LIN {X 116.831,Y -35.719,Z -65.842,A -90.000,B 90.000,C 0.000} C_DIS
LIN {X 116.119,Y -35.719,Z -68.117,A -90.000,B 90.000,C 0.000} C_DIS
LIN {X 115.340,Y -35.719,Z -70.370,A -90.000,B 90.000,C 0.000} C_DIS
LIN {X 114.495,Y -35.719,Z -72.600,A -90.000,B 90.000,C 0.000} C_DIS
LIN {X 113.585,Y -35.719,Z -74.804,A -90.000,B 90.000,C 0.000} C_DIS
LIN {X 112.611,Y -35.719,Z -76.980,A -90.000,B 90.000,C 0.000} C_DIS
LIN {X 111.574,Y -35.719,Z -79.127,A -90.000,B 90.000,C 0.000} C_DIS
LIN {X 110.474,Y -35.719,Z -81.243,A -90.000,B 90.000,C 0.000} C_DIS
LIN {X 109.313,Y -35.719,Z -83.325,A -90.000,B 90.000,C 0.000} C_DIS
LIN {X 108.091,Y -35.719,Z -85.373,A -90.000,B 90.000,C 0.000} C_DIS
LIN {X 106.810,Y -35.719,Z -87.384,A -90.000,B 90.000,C 0.000} C_DIS
LIN {X 105.470,Y -35.719,Z -89.356,A -90.000,B 90.000,C 0.000} C_DIS
LIN {X 105.415,Y -35.719,Z -90.221,A -90.000,B 90.000,C 0.000} C_DIS
LIN {X 105.339,Y -35.719,Z -91.084,A -90.000,B 90.000,C 0.000} C_DIS
LIN {X 105.322,Y -35.719,Z -92.275,A -90.000,B 90.000,C 0.000} C_DIS
LIN {X 105.256,Y -35.719,Z -93.465,A -90.000,B 90.000,C 0.000} C_DIS
LIN {X 105.138,Y -35.719,Z -94.651,A -90.000,B 90.000,C 0.000} C_DIS
LIN {X 104.971,Y -35.719,Z -95.830,A -90.000,B 90.000,C 0.000} C_DIS
LIN {X 104.754,Y -35.719,Z -97.002,A -90.000,B 90.000,C 0.000} C_DIS
LIN {X 104.487,Y -35.719,Z -98.163,A -90.000,B 90.000,C 0.000} C_DIS
LIN {X 104.172,Y -35.719,Z -99.312,A -90.000,B 90.000,C 0.000} C_DIS
LIN {X 103.843,Y -35.719,Z -100.216,A -90.000,B 90.000,C 0.000} C_DIS
LIN {X 103.553,Y -35.719,Z -101.134,A -90.000,B 90.000,C 0.000} C_DIS
LIN {X 103.303,Y -35.719,Z -102.064,A -90.000,B 90.000,C 0.000} C_DIS
LIN {X 103.095,Y -35.719,Z -103.004,A -90.000,B 90.000,C 0.000} C_DIS
LIN {X 102.892,Y -35.719,Z -103.459,A -90.000,B 90.000,C 0.000} C_DIS
LIN {X 102.749,Y -35.719,Z -103.936,A -90.000,B 90.000,C 0.000} C_DIS
LIN {X 102.667,Y -35.719,Z -104.427,A -90.000,B 90.000,C 0.000} C_DIS
LIN {X 102.649,Y -35.719,Z -104.925,A -90.000,B 90.000,C 0.000} C_DIS
LIN {X 102.693,Y -35.719,Z -105.421,A -90.000,B 90.000,C 0.000} C_DIS
LIN {X 102.800,Y -35.719,Z -105.907,A -90.000,B 90.000,C 0.000} C_DIS
LIN {X 102.981,Y -35.719,Z -108.478,A -90.000,B 90.000,C 0.000} C_DIS
LIN {X 103.102,Y -35.719,Z -111.053,A -90.000,B 90.000,C 0.000} C_DIS
LIN {X 103.163,Y -35.719,Z -113.630,A -90.000,B 90.000,C 0.000} C_DIS
LIN {X 103.164,Y -35.719,Z -116.208,A -90.000,B 90.000,C 0.000} C_DIS
LIN {X 103.250,Y -35.719,Z -118.970,A -90.000,B 90.000,C 0.000} C_DIS
LIN {X 103.278,Y -35.719,Z -121.732,A -90.000,B 90.000,C 0.000} C_DIS
LIN {X 103.247,Y -35.719,Z -124.495,A -90.000,B 90.000,C 0.000} C_DIS
LIN {X 103.157,Y -35.719,Z -127.257,A -90.000,B 90.000,C 0.000} C_DIS
LIN {X 103.009,Y -35.719,Z -130.016,A -90.000,B 90.000,C 0.000} C_DIS
LIN {X 102.803,Y -35.719,Z -132.771,A -90.000,B 90.000,C 0.000} C_DIS
LIN {X 102.538,Y -35.719,Z -135.521,A -90.000,B 90.000,C 0.000} C_DIS
LIN {X 102.366,Y -35.719,Z -138.398,A -90.000,B 90.000,C 0.000} C_DIS
LIN {X 102.141,Y -35.719,Z -141.271,A -90.000,B 90.000,C 0.000} C_DIS
LIN {X 101.862,Y -35.719,Z -144.140,A -90.000,B 90.000,C 0.000} C_DIS
LIN {X 101.529,Y -35.719,Z -147.003,A -90.000,B 90.000,C 0.000} C_DIS
LIN {X 101.143,Y -35.719,Z -149.859,A -90.000,B 90.000,C 0.000} C_DIS
LIN {X 100.704,Y -35.719,Z -152.708,A -90.000,B 90.000,C 0.000} C_DIS
LIN {X 100.212,Y -35.719,Z -155.548,A -90.000,B 90.000,C 0.000} C_DIS
LIN {X 99.667,Y -35.719,Z -158.378,A -90.000,B 90.000,C 0.000} C_DIS
LIN {X 98.834,Y -35.719,Z -161.929,A -90.000,B 90.000,C 0.000} C_DIS
LIN {X 97.948,Y -35.719,Z -165.466,A -90.000,B 90.000,C 0.000} C_DIS
LIN {X 97.008,Y -35.719,Z -168.990,A -90.000,B 90.000,C 0.000} C_DIS
LIN {X 96.014,Y -35.719,Z -172.499,A -90.000,B 90.000,C 0.000} C_DIS
LIN {X 94.967,Y -35.719,Z -175.992,A -90.000,B 90.000,C 0.000} C_DIS
LIN {X 93.867,Y -35.719,Z -179.469,A -90.000,B 90.000,C 0.000} C_DIS
LIN {X 89.622,Y -35.719,Z -192.770,A -90.000,B 90.000,C 0.000} C_DIS
LIN {X 88.034,Y -35.719,Z -197.593,A -90.000,B 90.000,C 0.000} C_DIS
LIN {X 86.382,Y -35.719,Z -202.396,A -90.000,B 90.000,C 0.000} C_DIS
LIN {X 84.667,Y -35.719,Z -207.176,A -90.000,B 90.000,C 0.000} C_DIS
LIN {X 82.889,Y -35.719,Z -211.933,A -90.000,B 90.000,C 0.000} C_DIS
LIN {X 81.049,Y -35.719,Z -216.666,A -90.000,B 90.000,C 0.000} C_DIS
LIN {X 79.146,Y -35.719,Z -221.374,A -90.000,B 90.000,C 0.000} C_DIS
LIN {X 76.777,Y -35.719,Z -226.893,A -90.000,B 90.000,C 0.000} C_DIS
LIN {X 74.453,Y -35.719,Z -232.431,A -90.000,B 90.000,C 0.000} C_DIS
LIN {X 72.173,Y -35.719,Z -237.987,A -90.000,B 90.000,C 0.000} C_DIS
LIN {X 69.938,Y -35.719,Z -243.561,A -90.000,B 90.000,C 0.000} C_DIS
LIN {X 145.015,Y -35.719,Z -243.561,A -90.000,B 90.000,C 0.000} C_DIS
LIN {X 145.015,Y -35.719,Z 0.000,A -90.000,B 90.000,C 0.000} C_DIS
LIN {X -145.015,Y -35.719,Z 0.000,A -90.000,B 90.000,C 0.000} C_DIS
LIN {X -145.015,Y -35.719,Z -243.561,A -90.000,B 90.000,C 0.000} C_DIS
LIN {X -110.096,Y -35.719,Z -243.561,A -90.000,B 90.000,C 0.000} C_DIS
LIN {X -107.153,Y -35.719,Z -241.272,A -90.000,B 90.000,C 0.000} C_DIS
LIN {X -104.176,Y -35.719,Z -239.027,A -90.000,B 90.000,C 0.000} C_DIS
LIN {X -101.166,Y -35.719,Z -236.828,A -90.000,B 90.000,C 0.000} C_DIS
LIN {X -98.123,Y -35.719,Z -234.673,A -90.000,B 90.000,C 0.000} C_DIS
LIN {X -95.049,Y -35.719,Z -232.564,A -90.000,B 90.000,C 0.000} C_DIS
LIN {X -91.943,Y -35.719,Z -230.501,A -90.000,B 90.000,C 0.000} C_DIS
LIN {X -88.807,Y -35.719,Z -228.485,A -90.000,B 90.000,C 0.000} C_DIS
LIN {X -86.159,Y -35.719,Z -226.746,A -90.000,B 90.000,C 0.000} C_DIS
LIN {X -81.987,Y -35.719,Z -224.226,A -90.000,B 90.000,C 0.000} C_DIS
LIN {X -77.783,Y -35.719,Z -221.761,A -90.000,B 90.000,C 0.000} C_DIS
LIN {X -73.548,Y -35.719,Z -219.350,A -90.000,B 90.000,C 0.000} C_DIS
LIN {X -69.281,Y -35.719,Z -216.994,A -90.000,B 90.000,C 0.000} C_DIS
LIN {X -64.985,Y -35.719,Z -214.693,A -90.000,B 90.000,C 0.000} C_DIS
LIN {X -60.659,Y -35.719,Z -212.448,A -90.000,B 90.000,C 0.000} C_DIS
LIN {X -56.305,Y -35.719,Z -210.259,A -90.000,B 90.000,C 0.000} C_DIS
LIN {X -51.922,Y -35.719,Z -208.127,A -90.000,B 90.000,C 0.000} C_DIS
LIN {X -46.937,Y -35.719,Z -205.632,A -90.000,B 90.000,C 0.000} C_DIS
LIN {X -44.461,Y -35.719,Z -204.434,A -90.000,B 90.000,C 0.000} C_DIS
LIN {X -42.009,Y -35.719,Z -203.189,A -90.000,B 90.000,C 0.000} C_DIS
LIN {X -39.581,Y -35.719,Z -201.895,A -90.000,B 90.000,C 0.000} C_DIS
LIN {X -37.180,Y -35.719,Z -200.555,A -90.000,B 90.000,C 0.000} C_DIS
LIN {X -34.804,Y -35.719,Z -199.168,A -90.000,B 90.000,C 0.000} C_DIS
LIN {X -32.457,Y -35.719,Z -197.735,A -90.000,B 90.000,C 0.000} C_DIS
LIN {X -30.138,Y -35.719,Z -196.256,A -90.000,B 90.000,C 0.000} C_DIS
LIN {X -27.848,Y -35.719,Z -194.732,A -90.000,B 90.000,C 0.000} C_DIS
LIN {X -24.879,Y -35.719,Z -192.551,A -90.000,B 90.000,C 0.000} C_DIS
LIN {X -21.945,Y -35.719,Z -190.324,A -90.000,B 90.000,C 0.000} C_DIS
LIN {X -19.046,Y -35.719,Z -188.051,A -90.000,B 90.000,C 0.000} C_DIS
LIN {X -16.183,Y -35.719,Z -185.732,A -90.000,B 90.000,C 0.000} C_DIS
LIN {X -13.358,Y -35.719,Z -183.368,A -90.000,B 90.000,C 0.000} C_DIS
LIN {X -10.570,Y -35.719,Z -180.960,A -90.000,B 90.000,C 0.000} C_DIS
LIN {X -7.820,Y -35.719,Z -178.509,A -90.000,B 90.000,C 0.000} C_DIS
LIN {X -5.995,Y -35.719,Z -176.907,A -90.000,B 90.000,C 0.000} C_DIS
LIN {X -4.209,Y -35.719,Z -175.263,A -90.000,B 90.000,C 0.000} C_DIS
LIN {X -2.461,Y -35.719,Z -173.577,A -90.000,B 90.000,C 0.000} C_DIS
LIN {X -0.754,Y -35.719,Z -171.851,A -90.000,B 90.000,C 0.000} C_DIS
LIN {X 0.913,Y -35.719,Z -170.085,A -90.000,B 90.000,C 0.000} C_DIS
LIN {X 1.496,Y -35.719,Z -169.467,A -90.000,B 90.000,C 0.000} C_DIS
LIN {X 2.036,Y -35.719,Z -168.811,A -90.000,B 90.000,C 0.000} C_DIS
LIN {X 2.530,Y -35.719,Z -168.120,A -90.000,B 90.000,C 0.000} C_DIS
LIN {X 2.976,Y -35.719,Z -167.397,A -90.000,B 90.000,C 0.000} C_DIS
LIN {X 3.229,Y -35.719,Z -167.142,A -90.000,B 90.000,C 0.000} C_DIS
LIN {X 3.431,Y -35.719,Z -166.845,A -90.000,B 90.000,C 0.000} C_DIS
LIN {X 3.574,Y -35.719,Z -166.515,A -90.000,B 90.000,C 0.000} C_DIS
LIN {X 3.653,Y -35.719,Z -166.164,A -90.000,B 90.000,C 0.000} C_DIS
LIN {X 3.666,Y -35.719,Z -165.805,A -90.000,B 90.000,C 0.000} C_DIS
LIN {X 3.612,Y -35.719,Z -165.450,A -90.000,B 90.000,C 0.000} C_DIS
LIN {X 3.493,Y -35.719,Z -165.111,A -90.000,B 90.000,C 0.000} C_DIS
LIN {X 3.313,Y -35.719,Z -164.800,A -90.000,B 90.000,C 0.000} C_DIS
LIN {X 3.078,Y -35.719,Z -164.528,A -90.000,B 90.000,C 0.000} C_DIS
LIN {X 2.322,Y -35.719,Z -164.113,A -90.000,B 90.000,C 0.000} C_DIS
LIN {X 1.554,Y -35.719,Z -163.721,A -90.000,B 90.000,C 0.000} C_DIS
LIN {X -1.251,Y -35.719,Z -162.907,A -90.000,B 90.000,C 0.000} C_DIS
LIN {X -2.477,Y -35.719,Z -162.410,A -90.000,B 90.000,C 0.000} C_DIS
LIN {X -3.719,Y -35.719,Z -161.957,A -90.000,B 90.000,C 0.000} C_DIS
LIN {X -4.976,Y -35.719,Z -161.547,A -90.000,B 90.000,C 0.000} C_DIS
LIN {X -6.247,Y -35.719,Z -161.182,A -90.000,B 90.000,C 0.000} C_DIS
LIN {X -8.359,Y -35.719,Z -160.357,A -90.000,B 90.000,C 0.000} C_DIS
LIN {X -10.450,Y -35.719,Z -159.479,A -90.000,B 90.000,C 0.000} C_DIS
LIN {X -12.518,Y -35.719,Z -158.548,A -90.000,B 90.000,C 0.000} C_DIS
LIN {X -14.562,Y -35.719,Z -157.566,A -90.000,B 90.000,C 0.000} C_DIS
LIN {X -16.580,Y -35.719,Z -156.532,A -90.000,B 90.000,C 0.000} C_DIS
LIN {X -18.572,Y -35.719,Z -155.448,A -90.000,B 90.000,C 0.000} C_DIS
LIN {X -20.770,Y -35.719,Z -154.028,A -90.000,B 90.000,C 0.000} C_DIS
LIN {X -22.940,Y -35.719,Z -152.565,A -90.000,B 90.000,C 0.000} C_DIS
LIN {X -25.081,Y -35.719,Z -151.060,A -90.000,B 90.000,C 0.000} C_DIS
LIN {X -27.192,Y -35.719,Z -149.513,A -90.000,B 90.000,C 0.000} C_DIS
LIN {X -28.258,Y -35.719,Z -148.710,A -90.000,B 90.000,C 0.000} C_DIS
LIN {X -29.291,Y -35.719,Z -147.865,A -90.000,B 90.000,C 0.000} C_DIS
LIN {X -30.291,Y -35.719,Z -146.981,A -90.000,B 90.000,C 0.000} C_DIS
LIN {X -31.255,Y -35.719,Z -146.058,A -90.000,B 90.000,C 0.000} C_DIS
LIN {X -32.182,Y -35.719,Z -145.098,A -90.000,B 90.000,C 0.000} C_DIS
LIN {X -33.529,Y -35.719,Z -143.805,A -90.000,B 90.000,C 0.000} C_DIS
LIN {X -34.823,Y -35.719,Z -142.460,A -90.000,B 90.000,C 0.000} C_DIS
LIN {X -36.063,Y -35.719,Z -141.064,A -90.000,B 90.000,C 0.000} C_DIS
LIN {X -37.246,Y -35.719,Z -139.620,A -90.000,B 90.000,C 0.000} C_DIS
LIN {X -38.372,Y -35.719,Z -138.130,A -90.000,B 90.000,C 0.000} C_DIS
LIN {X -39.437,Y -35.719,Z -136.597,A -90.000,B 90.000,C 0.000} C_DIS
LIN {X -40.440,Y -35.719,Z -135.022,A -90.000,B 90.000,C 0.000} C_DIS
LIN {X -41.380,Y -35.719,Z -133.409,A -90.000,B 90.000,C 0.000} C_DIS
LIN {X -42.255,Y -35.719,Z -131.760,A -90.000,B 90.000,C 0.000} C_DIS
LIN {X -43.063,Y -35.719,Z -130.077,A -90.000,B 90.000,C 0.000} C_DIS
LIN {X -43.805,Y -35.719,Z -128.364,A -90.000,B 90.000,C 0.000} C_DIS
LIN {X -44.477,Y -35.719,Z -126.622,A -90.000,B 90.000,C 0.000} C_DIS
LIN {X -45.080,Y -35.719,Z -124.855,A -90.000,B 90.000,C 0.000} C_DIS
LIN {X -45.612,Y -35.719,Z -123.065,A -90.000,B 90.000,C 0.000} C_DIS
LIN {X -46.072,Y -35.719,Z -121.256,A -90.000,B 90.000,C 0.000} C_DIS
LIN {X -46.455,Y -35.719,Z -119.310,A -90.000,B 90.000,C 0.000} C_DIS
LIN {X -46.782,Y -35.719,Z -117.354,A -90.000,B 90.000,C 0.000} C_DIS
LIN {X -47.053,Y -35.719,Z -115.390,A -90.000,B 90.000,C 0.000} C_DIS
LIN {X -47.268,Y -35.719,Z -113.418,A -90.000,B 90.000,C 0.000} C_DIS
LIN {X -47.426,Y -35.719,Z -111.441,A -90.000,B 90.000,C 0.000} C_DIS
LIN {X -47.529,Y -35.719,Z -109.461,A -90.000,B 90.000,C 0.000} C_DIS
LIN {X -47.947,Y -35.719,Z -108.832,A -90.000,B 90.000,C 0.000} C_DIS
LIN {X -48.399,Y -35.719,Z -108.227,A -90.000,B 90.000,C 0.000} C_DIS
LIN {X -48.883,Y -35.719,Z -107.647,A -90.000,B 90.000,C 0.000} C_DIS
LIN {X -50.094,Y -35.719,Z -106.124,A -90.000,B 90.000,C 0.000} C_DIS
LIN {X -51.246,Y -35.719,Z -104.556,A -90.000,B 90.000,C 0.000} C_DIS
LIN {X -52.339,Y -35.719,Z -102.947,A -90.000,B 90.000,C 0.000} C_DIS
LIN {X -53.372,Y -35.719,Z -101.298,A -90.000,B 90.000,C 0.000} C_DIS
LIN {X -54.341,Y -35.719,Z -99.611,A -90.000,B 90.000,C 0.000} C_DIS
LIN {X -55.247,Y -35.719,Z -97.889,A -90.000,B 90.000,C 0.000} C_DIS
LIN {X -56.088,Y -35.719,Z -96.135,A -90.000,B 90.000,C 0.000} C_DIS
LIN {X -56.863,Y -35.719,Z -94.350,A -90.000,B 90.000,C 0.000} C_DIS
LIN {X -57.570,Y -35.719,Z -92.538,A -90.000,B 90.000,C 0.000} C_DIS
LIN {X -58.209,Y -35.719,Z -90.700,A -90.000,B 90.000,C 0.000} C_DIS
LIN {X -58.779,Y -35.719,Z -88.840,A -90.000,B 90.000,C 0.000} C_DIS
LIN {X -59.279,Y -35.719,Z -86.960,A -90.000,B 90.000,C 0.000} C_DIS
LIN {X -59.708,Y -35.719,Z -85.062,A -90.000,B 90.000,C 0.000} C_DIS
LIN {X -60.066,Y -35.719,Z -83.149,A -90.000,B 90.000,C 0.000} C_DIS
LIN {X -60.352,Y -35.719,Z -81.225,A -90.000,B 90.000,C 0.000} C_DIS
LIN {X -60.530,Y -35.719,Z -79.874,A -90.000,B 90.000,C 0.000} C_DIS
LIN {X -60.643,Y -35.719,Z -78.516,A -90.000,B 90.000,C 0.000} C_DIS
LIN {X -60.688,Y -35.719,Z -77.155,A -90.000,B 90.000,C 0.000} C_DIS
LIN {X -60.667,Y -35.719,Z -75.792,A -90.000,B 90.000,C 0.000} C_DIS
LIN {X -60.578,Y -35.719,Z -74.433,A -90.000,B 90.000,C 0.000} C_DIS
LIN {X -60.424,Y -35.719,Z -73.079,A -90.000,B 90.000,C 0.000} C_DIS
LIN {X -60.203,Y -35.719,Z -71.734,A -90.000,B 90.000,C 0.000} C_DIS
LIN {X -59.916,Y -35.719,Z -70.402,A -90.000,B 90.000,C 0.000} C_DIS
LIN {X -59.565,Y -35.719,Z -69.086,A -90.000,B 90.000,C 0.000} C_DIS
LIN {X -59.313,Y -35.719,Z -68.078,A -90.000,B 90.000,C 0.000} C_DIS
LIN {X -58.993,Y -35.719,Z -67.089,A -90.000,B 90.000,C 0.000} C_DIS
LIN {X -58.606,Y -35.719,Z -66.124,A -90.000,B 90.000,C 0.000} C_DIS
LIN {X -58.155,Y -35.719,Z -65.188,A -90.000,B 90.000,C 0.000} C_DIS
LIN {X -57.640,Y -35.719,Z -64.284,A -90.000,B 90.000,C 0.000} C_DIS
LIN {X -57.066,Y -35.719,Z -63.418,A -90.000,B 90.000,C 0.000} C_DIS
LIN {X -56.434,Y -35.719,Z -62.593,A -90.000,B 90.000,C 0.000} C_DIS
LIN {X -55.747,Y -35.719,Z -61.813,A -90.000,B 90.000,C 0.000} C_DIS
LIN {X -55.009,Y -35.719,Z -61.081,A -90.000,B 90.000,C 0.000} C_DIS
LIN {X -54.222,Y -35.719,Z -60.402,A -90.000,B 90.000,C 0.000} C_DIS
LIN {X -53.391,Y -35.719,Z -59.777,A -90.000,B 90.000,C 0.000} C_DIS
LIN {X -52.520,Y -35.719,Z -59.210,A -90.000,B 90.000,C 0.000} C_DIS
LIN {X -51.321,Y -35.719,Z -58.559,A -90.000,B 90.000,C 0.000} C_DIS
LIN {X -50.096,Y -35.719,Z -57.960,A -90.000,B 90.000,C 0.000} C_DIS
LIN {X -48.846,Y -35.719,Z -57.414,A -90.000,B 90.000,C 0.000} C_DIS
LIN {X -47.573,Y -35.719,Z -56.922,A -90.000,B 90.000,C 0.000} C_DIS
LIN {X -46.281,Y -35.719,Z -56.485,A -90.000,B 90.000,C 0.000} C_DIS
LIN {X -44.691,Y -35.719,Z -56.129,A -90.000,B 90.000,C 0.000} C_DIS
LIN {X -43.088,Y -35.719,Z -55.836,A -90.000,B 90.000,C 0.000} C_DIS
LIN {X -41.475,Y -35.719,Z -55.608,A -90.000,B 90.000,C 0.000} C_DIS
LIN {X -39.854,Y -35.719,Z -55.444,A -90.000,B 90.000,C 0.000} C_DIS
LIN {X -38.227,Y -35.719,Z -55.345,A -90.000,B 90.000,C 0.000} C_DIS
LIN {X -36.598,Y -35.719,Z -55.310,A -90.000,B 90.000,C 0.000} C_DIS
LIN {X -34.969,Y -35.719,Z -55.340,A -90.000,B 90.000,C 0.000} C_DIS
LIN {X -33.343,Y -35.719,Z -55.435,A -90.000,B 90.000,C 0.000} C_DIS
LIN {X -31.721,Y -35.719,Z -55.595,A -90.000,B 90.000,C 0.000} C_DIS
LIN {X -30.107,Y -35.719,Z -55.819,A -90.000,B 90.000,C 0.000} C_DIS
LIN {X -28.504,Y -35.719,Z -56.107,A -90.000,B 90.000,C 0.000} C_DIS
LIN {X -26.913,Y -35.719,Z -56.459,A -90.000,B 90.000,C 0.000} C_DIS
LIN {X -25.337,Y -35.719,Z -56.874,A -90.000,B 90.000,C 0.000} C_DIS
LIN {X -25.206,Y -35.719,Z -56.732,A -90.000,B 90.000,C 0.000} C_DIS
LIN {X -24.358,Y -35.719,Z -56.061,A -90.000,B 90.000,C 0.000} C_DIS
LIN {X -23.471,Y -35.719,Z -55.444,A -90.000,B 90.000,C 0.000} C_DIS
LIN {X -22.548,Y -35.719,Z -54.882,A -90.000,B 90.000,C 0.000} C_DIS
LIN {X -21.592,Y -35.719,Z -54.378,A -90.000,B 90.000,C 0.000} C_DIS
LIN {X -20.607,Y -35.719,Z -53.933,A -90.000,B 90.000,C 0.000} C_DIS
LIN {X -19.596,Y -35.719,Z -53.549,A -90.000,B 90.000,C 0.000} C_DIS
LIN {X -18.564,Y -35.719,Z -53.229,A -90.000,B 90.000,C 0.000} C_DIS
LIN {X -17.514,Y -35.719,Z -52.972,A -90.000,B 90.000,C 0.000} C_DIS
LIN {X -16.196,Y -35.719,Z -52.825,A -90.000,B 90.000,C 0.000} C_DIS
LIN {X -14.873,Y -35.719,Z -52.731,A -90.000,B 90.000,C 0.000} C_DIS
LIN {X -13.548,Y -35.719,Z -52.688,A -90.000,B 90.000,C 0.000} C_DIS
LIN {X -12.222,Y -35.719,Z -52.697,A -90.000,B 90.000,C 0.000} C_DIS
LIN {X -10.897,Y -35.719,Z -52.757,A -90.000,B 90.000,C 0.000} C_DIS
LIN {X -9.576,Y -35.719,Z -52.870,A -90.000,B 90.000,C 0.000} C_DIS
LIN {X -8.260,Y -35.719,Z -53.034,A -90.000,B 90.000,C 0.000} C_DIS
LIN {X -4.666,Y -35.719,Z -53.602,A -90.000,B 90.000,C 0.000} C_DIS
LIN {X -1.066,Y -35.719,Z -54.121,A -90.000,B 90.000,C 0.000} C_DIS
LIN {X 2.542,Y -35.719,Z -54.591,A -90.000,B 90.000,C 0.000} C_DIS
LIN {X 2.542,Y -48.219,Z -54.591,A -90.000,B 90.000,C 0.000} C_DIS
LIN {X 2.542,Y -60.719,Z -54.591,A -90.000,B 90.000,C 0.000} C_DIS
LIN {X 90.609,Y -60.719,Z -242.561,A -90.000,B 90.000,C 0.000} C_DIS
LIN {X 90.609,Y -53.575,Z -242.561,A -90.000,B 90.000,C 0.000} C_DIS
LIN {X 90.609,Y -41.075,Z -242.561,A -90.000,B 90.000,C 0.000} C_DIS
LIN {X 90.609,Y -28.575,Z -242.561,A -90.000,B 90.000,C 0.000} C_DIS
LIN {X 144.015,Y -28.575,Z -242.561,A -90.000,B 90.000,C 0.000} C_DIS
LIN {X 144.015,Y -28.575,Z -235.012,A -90.000,B 90.000,C 0.000} C_DIS
LIN {X 92.953,Y -28.575,Z -235.012,A -90.000,B 90.000,C 0.000} C_DIS
LIN {X 93.660,Y -28.575,Z -232.505,A -90.000,B 90.000,C 0.000} C_DIS
LIN {X 94.335,Y -28.575,Z -229.989,A -90.000,B 90.000,C 0.000} C_DIS
LIN {X 94.978,Y -28.575,Z -227.464,A -90.000,B 90.000,C 0.000} C_DIS
LIN {X 144.015,Y -28.575,Z -227.464,A -90.000,B 90.000,C 0.000} C_DIS
LIN {X 144.015,Y -28.575,Z -219.915,A -90.000,B 90.000,C 0.000} C_DIS
LIN {X 96.864,Y -28.575,Z -219.915,A -90.000,B 90.000,C 0.000} C_DIS
LIN {X 97.478,Y -28.575,Z -217.548,A -90.000,B 90.000,C 0.000} C_DIS
LIN {X 98.098,Y -28.575,Z -215.183,A -90.000,B 90.000,C 0.000} C_DIS
LIN {X 98.477,Y -28.575,Z -213.776,A -90.000,B 90.000,C 0.000} C_DIS
LIN {X 98.848,Y -28.575,Z -212.366,A -90.000,B 90.000,C 0.000} C_DIS
LIN {X 144.015,Y -28.575,Z -212.366,A -90.000,B 90.000,C 0.000} C_DIS
LIN {X 144.015,Y -28.575,Z -204.817,A -90.000,B 90.000,C 0.000} C_DIS
LIN {X 100.664,Y -28.575,Z -204.817,A -90.000,B 90.000,C 0.000} C_DIS
LIN {X 101.185,Y -28.575,Z -202.411,A -90.000,B 90.000,C 0.000} C_DIS
LIN {X 101.679,Y -28.575,Z -200.000,A -90.000,B 90.000,C 0.000} C_DIS
LIN {X 102.147,Y -28.575,Z -197.583,A -90.000,B 90.000,C 0.000} C_DIS
LIN {X 102.190,Y -28.575,Z -197.269,A -90.000,B 90.000,C 0.000} C_DIS
LIN {X 144.015,Y -28.575,Z -197.269,A -90.000,B 90.000,C 0.000} C_DIS
LIN {X 144.015,Y -28.575,Z -189.720,A -90.000,B 90.000,C 0.000} C_DIS
LIN {X 102.994,Y -28.575,Z -189.720,A -90.000,B 90.000,C 0.000} C_DIS
LIN {X 103.117,Y -28.575,Z -188.042,A -90.000,B 90.000,C 0.000} C_DIS
LIN {X 103.220,Y -28.575,Z -186.362,A -90.000,B 90.000,C 0.000} C_DIS
LIN {X 103.302,Y -28.575,Z -184.681,A -90.000,B 90.000,C 0.000} C_DIS
LIN {X 103.398,Y -28.575,Z -183.426,A -90.000,B 90.000,C 0.000} C_DIS
LIN {X 103.504,Y -28.575,Z -182.171,A -90.000,B 90.000,C 0.000} C_DIS
LIN {X 144.015,Y -28.575,Z -182.171,A -90.000,B 90.000,C 0.000} C_DIS
LIN {X 144.015,Y -28.575,Z -174.622,A -90.000,B 90.000,C 0.000} C_DIS
LIN {X 104.367,Y -28.575,Z -174.622,A -90.000,B 90.000,C 0.000} C_DIS
LIN {X 104.655,Y -28.575,Z -172.656,A -90.000,B 90.000,C 0.000} C_DIS
LIN {X 104.969,Y -28.575,Z -170.694,A -90.000,B 90.000,C 0.000} C_DIS
LIN {X 105.308,Y -28.575,Z -168.736,A -90.000,B 90.000,C 0.000} C_DIS
LIN {X 105.494,Y -28.575,Z -167.073,A -90.000,B 90.000,C 0.000} C_DIS
LIN {X 144.015,Y -28.575,Z -167.073,A -90.000,B 90.000,C 0.000} C_DIS
LIN {X 144.015,Y -28.575,Z -159.525,A -90.000,B 90.000,C 0.000} C_DIS
LIN {X 106.509,Y -28.575,Z -159.525,A -90.000,B 90.000,C 0.000} C_DIS
LIN {X 106.823,Y -28.575,Z -157.546,A -90.000,B 90.000,C 0.000} C_DIS
LIN {X 107.130,Y -28.575,Z -154.760,A -90.000,B 90.000,C 0.000} C_DIS
LIN {X 107.450,Y -28.575,Z -151.976,A -90.000,B 90.000,C 0.000} C_DIS
LIN {X 144.015,Y -28.575,Z -151.976,A -90.000,B 90.000,C 0.000} C_DIS
LIN {X 144.015,Y -28.575,Z -144.427,A -90.000,B 90.000,C 0.000} C_DIS
LIN {X 108.180,Y -28.575,Z -144.427,A -90.000,B 90.000,C 0.000} C_DIS
LIN {X 108.464,Y -28.575,Z -140.654,A -90.000,B 90.000,C 0.000} C_DIS
LIN {X 108.704,Y -28.575,Z -136.878,A -90.000,B 90.000,C 0.000} C_DIS
LIN {X 144.015,Y -28.575,Z -136.878,A -90.000,B 90.000,C 0.000} C_DIS
LIN {X 144.015,Y -28.575,Z -129.329,A -90.000,B 90.000,C 0.000} C_DIS
LIN {X 109.051,Y -28.575,Z -129.329,A -90.000,B 90.000,C 0.000} C_DIS
LIN {X 109.121,Y -28.575,Z -127.065,A -90.000,B 90.000,C 0.000} C_DIS
LIN {X 109.176,Y -28.575,Z -124.801,A -90.000,B 90.000,C 0.000} C_DIS
LIN {X 109.139,Y -28.575,Z -123.291,A -90.000,B 90.000,C 0.000} C_DIS
LIN {X 109.089,Y -28.575,Z -121.781,A -90.000,B 90.000,C 0.000} C_DIS
LIN {X 144.015,Y -28.575,Z -121.781,A -90.000,B 90.000,C 0.000} C_DIS
LIN {X 144.015,Y -28.575,Z -114.232,A -90.000,B 90.000,C 0.000} C_DIS
LIN {X 108.661,Y -28.575,Z -114.232,A -90.000,B 90.000,C 0.000} C_DIS
LIN {X 108.444,Y -28.575,Z -111.646,A -90.000,B 90.000,C 0.000} C_DIS
LIN {X 108.192,Y -28.575,Z -109.064,A -90.000,B 90.000,C 0.000} C_DIS
LIN {X 108.100,Y -28.575,Z -107.872,A -90.000,B 90.000,C 0.000} C_DIS
LIN {X 107.977,Y -28.575,Z -106.683,A -90.000,B 90.000,C 0.000} C_DIS
LIN {X 144.015,Y -28.575,Z -106.683,A -90.000,B 90.000,C 0.000} C_DIS
LIN {X 144.015,Y -28.575,Z -99.134,A -90.000,B 90.000,C 0.000} C_DIS
LIN {X 107.607,Y -28.575,Z -99.134,A -90.000,B 90.000,C 0.000} C_DIS
LIN {X 107.662,Y -28.575,Z -98.377,A -90.000,B 90.000,C 0.000} C_DIS
LIN {X 107.727,Y -28.575,Z -97.620,A -90.000,B 90.000,C 0.000} C_DIS
LIN {X 107.725,Y -28.575,Z -97.442,A -90.000,B 90.000,C 0.000} C_DIS
LIN {X 107.818,Y -28.575,Z -95.980,A -90.000,B 90.000,C 0.000} C_DIS
LIN {X 107.875,Y -28.575,Z -94.516,A -90.000,B 90.000,C 0.000} C_DIS
LIN {X 107.894,Y -28.575,Z -93.051,A -90.000,B 90.000,C 0.000} C_DIS
LIN {X 107.877,Y -28.575,Z -91.586,A -90.000,B 90.000,C 0.000} C_DIS
LIN {X 144.015,Y -28.575,Z -91.586,A -90.000,B 90.000,C 0.000} C_DIS
LIN {X 144.015,Y -28.575,Z -84.037,A -90.000,B 90.000,C 0.000} C_DIS
LIN {X 110.095,Y -28.575,Z -84.037,A -90.000,B 90.000,C 0.000} C_DIS
LIN {X 111.154,Y -28.575,Z -82.191,A -90.000,B 90.000,C 0.000} C_DIS
LIN {X 112.160,Y -28.575,Z -80.317,A -90.000,B 90.000,C 0.000} C_DIS
LIN {X 113.115,Y -28.575,Z -78.416,A -90.000,B 90.000,C 0.000} C_DIS
LIN {X 114.015,Y -28.575,Z -76.488,A -90.000,B 90.000,C 0.000} C_DIS
LIN {X 144.015,Y -28.575,Z -76.488,A -90.000,B 90.000,C 0.000} C_DIS
LIN {X 144.015,Y -28.575,Z -68.939,A -90.000,B 90.000,C 0.000} C_DIS
LIN {X 116.946,Y -28.575,Z -68.939,A -90.000,B 90.000,C 0.000} C_DIS
LIN {X 117.479,Y -28.575,Z -67.249,A -90.000,B 90.000,C 0.000} C_DIS
LIN {X 117.973,Y -28.575,Z -65.548,A -90.000,B 90.000,C 0.000} C_DIS
LIN {X 118.427,Y -28.575,Z -63.835,A -90.000,B 90.000,C 0.000} C_DIS
LIN {X 118.842,Y -28.575,Z -62.113,A -90.000,B 90.000,C 0.000} C_DIS
LIN {X 119.052,Y -28.575,Z -61.390,A -90.000,B 90.000,C 0.000} C_DIS
LIN {X 144.015,Y -28.575,Z -61.390,A -90.000,B 90.000,C 0.000} C_DIS
LIN {X 144.015,Y -28.575,Z -53.842,A -90.000,B 90.000,C 0.000} C_DIS
LIN {X 122.255,Y -28.575,Z -53.842,A -90.000,B 90.000,C 0.000} C_DIS
LIN {X 122.641,Y -28.575,Z -53.168,A -90.000,B 90.000,C 0.000} C_DIS
LIN {X 123.155,Y -28.575,Z -52.067,A -90.000,B 90.000,C 0.000} C_DIS
LIN {X 123.623,Y -28.575,Z -50.946,A -90.000,B 90.000,C 0.000} C_DIS
LIN {X 124.043,Y -28.575,Z -49.806,A -90.000,B 90.000,C 0.000} C_DIS
LIN {X 124.414,Y -28.575,Z -48.649,A -90.000,B 90.000,C 0.000} C_DIS
LIN {X 124.736,Y -28.575,Z -47.477,A -90.000,B 90.000,C 0.000} C_DIS
LIN {X 125.008,Y -28.575,Z -46.293,A -90.000,B 90.000,C 0.000} C_DIS
LIN {X 144.015,Y -28.575,Z -46.293,A -90.000,B 90.000,C 0.000} C_DIS
LIN {X 144.015,Y -28.575,Z -38.744,A -90.000,B 90.000,C 0.000} C_DIS
LIN {X 124.956,Y -28.575,Z -38.744,A -90.000,B 90.000,C 0.000} C_DIS
LIN {X 124.685,Y -28.575,Z -37.760,A -90.000,B 90.000,C 0.000} C_DIS
LIN {X 124.354,Y -28.575,Z -36.794,A -90.000,B 90.000,C 0.000} C_DIS
LIN {X 123.965,Y -28.575,Z -35.849,A -90.000,B 90.000,C 0.000} C_DIS
LIN {X 123.520,Y -28.575,Z -34.931,A -90.000,B 90.000,C 0.000} C_DIS
LIN {X 123.019,Y -28.575,Z -34.041,A -90.000,B 90.000,C 0.000} C_DIS
LIN {X 122.465,Y -28.575,Z -33.183,A -90.000,B 90.000,C 0.000} C_DIS
LIN {X 121.880,Y -28.575,Z -32.488,A -90.000,B 90.000,C 0.000} C_DIS
LIN {X 121.259,Y -28.575,Z -31.825,A -90.000,B 90.000,C 0.000} C_DIS
LIN {X 120.604,Y -28.575,Z -31.195,A -90.000,B 90.000,C 0.000} C_DIS
LIN {X 144.015,Y -28.575,Z -31.195,A -90.000,B 90.000,C 0.000} C_DIS
LIN {X 144.015,Y -28.575,Z -23.646,A -90.000,B 90.000,C 0.000} C_DIS
LIN {X -144.015,Y -28.575,Z -23.646,A -90.000,B 90.000,C 0.000} C_DIS
LIN {X -144.015,Y -28.575,Z -16.098,A -90.000,B 90.000,C 0.000} C_DIS
LIN {X 144.015,Y -28.575,Z -16.098,A -90.000,B 90.000,C 0.000} C_DIS
LIN {X 144.015,Y -28.575,Z -8.549,A -90.000,B 90.000,C 0.000} C_DIS
LIN {X -144.015,Y -28.575,Z -8.549,A -90.000,B 90.000,C 0.000} C_DIS
LIN {X -144.015,Y -28.575,Z -1.000,A -90.000,B 90.000,C 0.000} C_DIS
LIN {X 144.015,Y -28.575,Z -1.000,A -90.000,B 90.000,C 0.000} C_DIS
LIN {X 98.289,Y -28.575,Z -31.195,A -90.000,B 90.000,C 0.000} C_DIS
LIN {X -144.015,Y -28.575,Z -31.195,A -90.000,B 90.000,C 0.000} C_DIS
LIN {X -144.015,Y -28.575,Z -38.744,A -90.000,B 90.000,C 0.000} C_DIS
LIN {X -101.193,Y -28.575,Z -38.744,A -90.000,B 90.000,C 0.000} C_DIS
LIN {X -101.596,Y -28.575,Z -39.028,A -90.000,B 90.000,C 0.000} C_DIS
LIN {X -101.986,Y -28.575,Z -39.330,A -90.000,B 90.000,C 0.000} C_DIS
LIN {X -102.094,Y -28.575,Z -39.429,A -90.000,B 90.000,C 0.000} C_DIS
LIN {X -102.751,Y -28.575,Z -39.948,A -90.000,B 90.000,C 0.000} C_DIS
LIN {X -103.368,Y -28.575,Z -40.513,A -90.000,B 90.000,C 0.000} C_DIS
LIN {X -103.943,Y -28.575,Z -41.121,A -90.000,B 90.000,C 0.000} C_DIS
LIN {X -104.473,Y -28.575,Z -41.768,A -90.000,B 90.000,C 0.000} C_DIS
LIN {X -104.954,Y -28.575,Z -42.453,A -90.000,B 90.000,C 0.000} C_DIS
LIN {X -105.385,Y -28.575,Z -43.170,A -90.000,B 90.000,C 0.000} C_DIS
LIN {X -105.763,Y -28.575,Z -43.917,A -90.000,B 90.000,C 0.000} C_DIS
LIN {X -106.085,Y -28.575,Z -44.689,A -90.000,B 90.000,C 0.000} C_DIS
LIN {X -106.352,Y -28.575,Z -45.483,A -90.000,B 90.000,C 0.000} C_DIS
LIN {X -106.560,Y -28.575,Z -46.293,A -90.000,B 90.000,C 0.000} C_DIS
LIN {X -144.015,Y -28.575,Z -46.293,A -90.000,B 90.000,C 0.000} C_DIS
LIN {X -144.015,Y -28.575,Z -53.842,A -90.000,B 90.000,C 0.000} C_DIS
LIN {X -106.161,Y -28.575,Z -53.842,A -90.000,B 90.000,C 0.000} C_DIS
LIN {X -105.911,Y -28.575,Z -54.488,A -90.000,B 90.000,C 0.000} C_DIS
LIN {X -105.627,Y -28.575,Z -55.119,A -90.000,B 90.000,C 0.000} C_DIS
LIN {X -105.310,Y -28.575,Z -55.735,A -90.000,B 90.000,C 0.000} C_DIS
LIN {X -104.928,Y -28.575,Z -56.497,A -90.000,B 90.000,C 0.000} C_DIS
LIN {X -104.507,Y -28.575,Z -57.239,A -90.000,B 90.000,C 0.000} C_DIS
LIN {X -104.048,Y -28.575,Z -57.957,A -90.000,B 90.000,C 0.000} C_DIS
LIN {X -103.552,Y -28.575,Z -58.651,A -90.000,B 90.000,C 0.000} C_DIS
LIN {X -103.021,Y -28.575,Z -59.318,A -90.000,B 90.000,C 0.000} C_DIS
LIN {X -102.889,Y -28.575,Z -59.474,A -90.000,B 90.000,C 0.000} C_DIS
LIN {X -102.004,Y -28.575,Z -60.445,A -90.000,B 90.000,C 0.000} C_DIS
LIN {X -101.092,Y -28.575,Z -61.390,A -90.000,B 90.000,C 0.000} C_DIS
LIN {X -144.015,Y -28.575,Z -61.390,A -90.000,B 90.000,C 0.000} C_DIS
LIN {X -144.015,Y -28.575,Z -68.939,A -90.000,B 90.000,C 0.000} C_DIS
LIN {X -94.433,Y -28.575,Z -68.939,A -90.000,B 90.000,C 0.000} C_DIS
LIN {X -93.947,Y -28.575,Z -69.354,A -90.000,B 90.000,C 0.000} C_DIS
LIN {X -93.454,Y -28.575,Z -69.760,A -90.000,B 90.000,C 0.000} C_DIS
LIN {X -93.308,Y -28.575,Z -70.531,A -90.000,B 90.000,C 0.000} C_DIS
LIN {X -93.115,Y -28.575,Z -71.292,A -90.000,B 90.000,C 0.000} C_DIS
LIN {X -92.875,Y -28.575,Z -72.040,A -90.000,B 90.000,C 0.000} C_DIS
LIN {X -92.588,Y -28.575,Z -72.771,A -90.000,B 90.000,C 0.000} C_DIS
LIN {X -92.257,Y -28.575,Z -73.482,A -90.000,B 90.000,C 0.000} C_DIS
LIN {X -91.882,Y -28.575,Z -74.172,A -90.000,B 90.000,C 0.000} C_DIS
LIN {X -91.423,Y -28.575,Z -74.970,A -90.000,B 90.000,C 0.000} C_DIS
LIN {X -90.924,Y -28.575,Z -75.742,A -90.000,B 90.000,C 0.000} C_DIS
LIN {X -90.385,Y -28.575,Z -76.488,A -90.000,B 90.000,C 0.000} C_DIS
LIN {X -144.015,Y -28.575,Z -76.488,A -90.000,B 90.000,C 0.000} C_DIS
LIN {X -144.015,Y -28.575,Z -84.037,A -90.000,B 90.000,C 0.000} C_DIS
LIN {X -77.948,Y -28.575,Z -84.037,A -90.000,B 90.000,C 0.000} C_DIS
LIN {X -76.119,Y -28.575,Z -85.996,A -90.000,B 90.000,C 0.000} C_DIS
LIN {X -74.283,Y -28.575,Z -87.949,A -90.000,B 90.000,C 0.000} C_DIS
LIN {X -72.604,Y -28.575,Z -89.776,A -90.000,B 90.000,C 0.000} C_DIS
LIN {X -70.908,Y -28.575,Z -91.586,A -90.000,B 90.000,C 0.000} C_DIS
LIN {X -144.015,Y -28.575,Z -91.586,A -90.000,B 90.000,C 0.000} C_DIS
LIN {X -144.015,Y -28.575,Z -99.134,A -90.000,B 90.000,C 0.000} C_DIS
LIN {X -64.714,Y -28.575,Z -99.134,A -90.000,B 90.000,C 0.000} C_DIS
LIN {X -63.497,Y -28.575,Z -100.750,A -90.000,B 90.000,C 0.000} C_DIS
LIN {X -62.304,Y -28.575,Z -102.383,A -90.000,B 90.000,C 0.000} C_DIS
LIN {X -61.134,Y -28.575,Z -104.033,A -90.000,B 90.000,C 0.000} C_DIS
LIN {X -60.125,Y -28.575,Z -105.362,A -90.000,B 90.000,C 0.000} C_DIS
LIN {X -59.107,Y -28.575,Z -106.683,A -90.000,B 90.000,C 0.000} C_DIS
LIN {X -144.015,Y -28.575,Z -106.683,A -90.000,B 90.000,C 0.000} C_DIS
LIN {X -144.015,Y -28.575,Z -114.232,A -90.000,B 90.000,C 0.000} C_DIS
LIN {X -53.346,Y -28.575,Z -114.232,A -90.000,B 90.000,C 0.000} C_DIS
LIN {X -52.039,Y -28.575,Z -116.132,A -90.000,B 90.000,C 0.000} C_DIS
LIN {X -50.773,Y -28.575,Z -118.060,A -90.000,B 90.000,C 0.000} C_DIS
LIN {X -49.551,Y -28.575,Z -120.015,A -90.000,B 90.000,C 0.000} C_DIS
LIN {X -48.708,Y -28.575,Z -121.781,A -90.000,B 90.000,C 0.000} C_DIS
LIN {X -144.015,Y -28.575,Z -121.781,A -90.000,B 90.000,C 0.000} C_DIS
LIN {X -144.015,Y -28.575,Z -129.329,A -90.000,B 90.000,C 0.000} C_DIS
LIN {X -45.193,Y -28.575,Z -129.329,A -90.000,B 90.000,C 0.000} C_DIS
LIN {X -44.370,Y -28.575,Z -130.880,A -90.000,B 90.000,C 0.000} C_DIS
LIN {X -43.511,Y -28.575,Z -132.411,A -90.000,B 90.000,C 0.000} C_DIS
LIN {X -42.616,Y -28.575,Z -133.921,A -90.000,B 90.000,C 0.000} C_DIS
LIN {X -41.687,Y -28.575,Z -135.411,A -90.000,B 90.000,C 0.000} C_DIS
LIN {X -40.723,Y -28.575,Z -136.878,A -90.000,B 90.000,C 0.000} C_DIS
LIN {X -144.015,Y -28.575,Z -136.878,A -90.000,B 90.000,C 0.000} C_DIS
LIN {X -144.015,Y -28.575,Z -144.427,A -90.000,B 90.000,C 0.000} C_DIS
LIN {X -35.127,Y -28.575,Z -144.427,A -90.000,B 90.000,C 0.000} C_DIS
LIN {X -33.918,Y -28.575,Z -145.910,A -90.000,B 90.000,C 0.000} C_DIS
LIN {X -32.661,Y -28.575,Z -147.353,A -90.000,B 90.000,C 0.000} C_DIS
LIN {X -31.357,Y -28.575,Z -148.754,A -90.000,B 90.000,C 0.000} C_DIS
LIN {X -30.008,Y -28.575,Z -150.111,A -90.000,B 90.000,C 0.000} C_DIS
LIN {X -28.615,Y -28.575,Z -151.423,A -90.000,B 90.000,C 0.000} C_DIS
LIN {X -28.018,Y -28.575,Z -151.976,A -90.000,B 90.000,C 0.000} C_DIS
LIN {X -144.015,Y -28.575,Z -151.976,A -90.000,B 90.000,C 0.000} C_DIS
LIN {X -144.015,Y -28.575,Z -159.525,A -90.000,B 90.000,C 0.000} C_DIS
LIN {X -19.165,Y -28.575,Z -159.525,A -90.000,B 90.000,C 0.000} C_DIS
LIN {X -17.121,Y -28.575,Z -161.109,A -90.000,B 90.000,C 0.000} C_DIS
LIN {X -15.051,Y -28.575,Z -162.658,A -90.000,B 90.000,C 0.000} C_DIS
LIN {X -13.519,Y -28.575,Z -163.850,A -90.000,B 90.000,C 0.000} C_DIS
LIN {X -12.006,Y -28.575,Z -165.066,A -90.000,B 90.000,C 0.000} C_DIS
LIN {X -12.135,Y -28.575,Z -165.743,A -90.000,B 90.000,C 0.000} C_DIS
LIN {X -12.297,Y -28.575,Z -166.412,A -90.000,B 90.000,C 0.000} C_DIS
LIN {X -12.492,Y -28.575,Z -167.073,A -90.000,B 90.000,C 0.000} C_DIS
LIN {X -144.015,Y -28.575,Z -167.073,A -90.000,B 90.000,C 0.000} C_DIS
LIN {X -144.015,Y -28.575,Z -174.622,A -90.000,B 90.000,C 0.000} C_DIS
LIN {X -16.782,Y -28.575,Z -174.622,A -90.000,B 90.000,C 0.000} C_DIS
LIN {X -17.686,Y -28.575,Z -175.838,A -90.000,B 90.000,C 0.000} C_DIS
LIN {X -18.627,Y -28.575,Z -177.025,A -90.000,B 90.000,C 0.000} C_DIS
LIN {X -19.603,Y -28.575,Z -178.184,A -90.000,B 90.000,C 0.000} C_DIS
LIN {X -20.614,Y -28.575,Z -179.312,A -90.000,B 90.000,C 0.000} C_DIS
LIN {X -21.659,Y -28.575,Z -180.409,A -90.000,B 90.000,C 0.000} C_DIS
LIN {X -22.737,Y -28.575,Z -181.474,A -90.000,B 90.000,C 0.000} C_DIS
LIN {X -23.420,Y -28.575,Z -182.171,A -90.000,B 90.000,C 0.000} C_DIS
LIN {X -144.015,Y -28.575,Z -182.171,A -90.000,B 90.000,C 0.000} C_DIS
LIN {X -144.015,Y -28.575,Z -189.720,A -90.000,B 90.000,C 0.000} C_DIS
LIN {X -32.227,Y -28.575,Z -189.720,A -90.000,B 90.000,C 0.000} C_DIS
LIN {X -33.745,Y -28.575,Z -190.794,A -90.000,B 90.000,C 0.000} C_DIS
LIN {X -35.291,Y -28.575,Z -191.829,A -90.000,B 90.000,C 0.000} C_DIS
LIN {X -36.862,Y -28.575,Z -192.823,A -90.000,B 90.000,C 0.000} C_DIS
LIN {X -38.458,Y -28.575,Z -193.777,A -90.000,B 90.000,C 0.000} C_DIS
LIN {X -40.079,Y -28.575,Z -194.690,A -90.000,B 90.000,C 0.000} C_DIS
LIN {X -42.260,Y -28.575,Z -195.983,A -90.000,B 90.000,C 0.000} C_DIS
LIN {X -44.445,Y -28.575,Z -197.269,A -90.000,B 90.000,C 0.000} C_DIS
LIN {X -144.015,Y -28.575,Z -197.269,A -90.000,B 90.000,C 0.000} C_DIS
LIN {X -144.015,Y -28.575,Z -204.817,A -90.000,B 90.000,C 0.000} C_DIS
LIN {X -57.587,Y -28.575,Z -204.817,A -90.000,B 90.000,C 0.000} C_DIS
LIN {X -64.145,Y -28.575,Z -208.574,A -90.000,B 90.000,C 0.000} C_DIS
LIN {X -70.660,Y -28.575,Z -212.366,A -90.000,B 90.000,C 0.000} C_DIS
LIN {X -144.015,Y -28.575,Z -212.366,A -90.000,B 90.000,C 0.000} C_DIS
LIN {X -144.015,Y -28.575,Z -219.915,A -90.000,B 90.000,C 0.000} C_DIS
LIN {X -83.257,Y -28.575,Z -219.915,A -90.000,B 90.000,C 0.000} C_DIS
LIN {X -87.261,Y -28.575,Z -222.401,A -90.000,B 90.000,C 0.000} C_DIS
LIN {X -91.247,Y -28.575,Z -224.917,A -90.000,B 90.000,C 0.000} C_DIS
LIN {X -95.213,Y -28.575,Z -227.464,A -90.000,B 90.000,C 0.000} C_DIS
LIN {X -144.015,Y -28.575,Z -227.464,A -90.000,B 90.000,C 0.000} C_DIS
LIN {X -144.015,Y -28.575,Z -235.012,A -90.000,B 90.000,C 0.000} C_DIS
LIN {X -106.598,Y -28.575,Z -235.012,A -90.000,B 90.000,C 0.000} C_DIS
LIN {X -110.238,Y -28.575,Z -237.503,A -90.000,B 90.000,C 0.000} C_DIS
LIN {X -113.861,Y -28.575,Z -240.019,A -90.000,B 90.000,C 0.000} C_DIS
LIN {X -117.466,Y -28.575,Z -242.561,A -90.000,B 90.000,C 0.000} C_DIS
LIN {X -144.015,Y -28.575,Z -242.561,A -90.000,B 90.000,C 0.000} C_DIS
LIN {X -77.047,Y -28.575,Z -85.003,A -90.000,B 90.000,C 0.000} C_DIS
LIN {X -78.629,Y -28.575,Z -83.304,A -90.000,B 90.000,C 0.000} C_DIS
LIN {X -79.728,Y -28.575,Z -83.123,A -90.000,B 90.000,C 0.000} C_DIS
LIN {X -80.813,Y -28.575,Z -82.873,A -90.000,B 90.000,C 0.000} C_DIS
LIN {X -81.880,Y -28.575,Z -82.556,A -90.000,B 90.000,C 0.000} C_DIS
LIN {X -82.926,Y -28.575,Z -82.172,A -90.000,B 90.000,C 0.000} C_DIS
LIN {X -83.945,Y -28.575,Z -81.723,A -90.000,B 90.000,C 0.000} C_DIS
LIN {X -84.934,Y -28.575,Z -81.212,A -90.000,B 90.000,C 0.000} C_DIS
LIN {X -85.889,Y -28.575,Z -80.639,A -90.000,B 90.000,C 0.000} C_DIS
LIN {X -86.806,Y -28.575,Z -80.007,A -90.000,B 90.000,C 0.000} C_DIS
LIN {X -87.681,Y -28.575,Z -79.318,A -90.000,B 90.000,C 0.000} C_DIS
LIN {X -88.512,Y -28.575,Z -78.577,A -90.000,B 90.000,C 0.000} C_DIS
LIN {X -89.294,Y -28.575,Z -77.784,A -90.000,B 90.000,C 0.000} C_DIS
LIN {X -90.025,Y -28.575,Z -76.944,A -90.000,B 90.000,C 0.000} C_DIS
LIN {X -90.702,Y -28.575,Z -76.059,A -90.000,B 90.000,C 0.000} C_DIS
LIN {X -91.322,Y -28.575,Z -75.134,A -90.000,B 90.000,C 0.000} C_DIS
LIN {X -91.882,Y -28.575,Z -74.172,A -90.000,B 90.000,C 0.000} C_DIS
LIN {X -92.257,Y -28.575,Z -73.482,A -90.000,B 90.000,C 0.000} C_DIS
LIN {X -92.588,Y -28.575,Z -72.771,A -90.000,B 90.000,C 0.000} C_DIS
LIN {X -92.875,Y -28.575,Z -72.040,A -90.000,B 90.000,C 0.000} C_DIS
LIN {X -93.115,Y -28.575,Z -71.292,A -90.000,B 90.000,C 0.000} C_DIS
LIN {X -93.309,Y -28.575,Z -70.531,A -90.000,B 90.000,C 0.000} C_DIS
LIN {X -93.454,Y -28.575,Z -69.760,A -90.000,B 90.000,C 0.000} C_DIS
LIN {X -94.309,Y -28.575,Z -69.047,A -90.000,B 90.000,C 0.000} C_DIS
LIN {X -95.141,Y -28.575,Z -68.308,A -90.000,B 90.000,C 0.000} C_DIS
LIN {X -95.290,Y -28.575,Z -68.169,A -90.000,B 90.000,C 0.000} C_DIS
LIN {X -95.872,Y -28.575,Z -67.573,A -90.000,B 90.000,C 0.000} C_DIS
LIN {X -96.415,Y -28.575,Z -66.941,A -90.000,B 90.000,C 0.000} C_DIS
LIN {X -96.917,Y -28.575,Z -66.275,A -90.000,B 90.000,C 0.000} C_DIS
LIN {X -97.376,Y -28.575,Z -65.580,A -90.000,B 90.000,C 0.000} C_DIS
LIN {X -97.790,Y -28.575,Z -64.856,A -90.000,B 90.000,C 0.000} C_DIS
LIN {X -98.157,Y -28.575,Z -64.108,A -90.000,B 90.000,C 0.000} C_DIS
LIN {X -99.400,Y -28.575,Z -63.013,A -90.000,B 90.000,C 0.000} C_DIS
LIN {X -100.604,Y -28.575,Z -61.874,A -90.000,B 90.000,C 0.000} C_DIS
LIN {X -101.768,Y -28.575,Z -60.694,A -90.000,B 90.000,C 0.000} C_DIS
LIN {X -102.889,Y -28.575,Z -59.474,A -90.000,B 90.000,C 0.000} C_DIS
LIN {X -103.021,Y -28.575,Z -59.318,A -90.000,B 90.000,C 0.000} C_DIS
LIN {X -103.552,Y -28.575,Z -58.651,A -90.000,B 90.000,C 0.000} C_DIS
LIN {X -104.048,Y -28.575,Z -57.957,A -90.000,B 90.000,C 0.000} C_DIS
LIN {X -104.507,Y -28.575,Z -57.239,A -90.000,B 90.000,C 0.000} C_DIS
LIN {X -104.928,Y -28.575,Z -56.497,A -90.000,B 90.000,C 0.000} C_DIS
LIN {X -105.310,Y -28.575,Z -55.735,A -90.000,B 90.000,C 0.000} C_DIS
LIN {X -105.709,Y -28.575,Z -54.945,A -90.000,B 90.000,C 0.000} C_DIS
LIN {X -106.054,Y -28.575,Z -54.130,A -90.000,B 90.000,C 0.000} C_DIS
LIN {X -106.343,Y -28.575,Z -53.293,A -90.000,B 90.000,C 0.000} C_DIS
LIN {X -106.575,Y -28.575,Z -52.439,A -90.000,B 90.000,C 0.000} C_DIS
LIN {X -106.748,Y -28.575,Z -51.570,A -90.000,B 90.000,C 0.000} C_DIS
LIN {X -106.861,Y -28.575,Z -50.693,A -90.000,B 90.000,C 0.000} C_DIS
LIN {X -106.915,Y -28.575,Z -49.809,A -90.000,B 90.000,C 0.000} C_DIS
LIN {X -106.909,Y -28.575,Z -48.924,A -90.000,B 90.000,C 0.000} C_DIS
LIN {X -106.843,Y -28.575,Z -48.041,A -90.000,B 90.000,C 0.000} C_DIS
LIN {X -106.716,Y -28.575,Z -47.165,A -90.000,B 90.000,C 0.000} C_DIS
LIN {X -106.569,Y -28.575,Z -46.337,A -90.000,B 90.000,C 0.000} C_DIS
LIN {X -106.363,Y -28.575,Z -45.521,A -90.000,B 90.000,C 0.000} C_DIS
LIN {X -106.098,Y -28.575,Z -44.723,A -90.000,B 90.000,C 0.000} C_DIS
LIN {X -105.776,Y -28.575,Z -43.945,A -90.000,B 90.000,C 0.000} C_DIS
LIN {X -105.398,Y -28.575,Z -43.194,A -90.000,B 90.000,C 0.000} C_DIS
LIN {X -104.966,Y -28.575,Z -42.472,A -90.000,B 90.000,C 0.000} C_DIS
LIN {X -104.484,Y -28.575,Z -41.783,A -90.000,B 90.000,C 0.000} C_DIS
LIN {X -103.952,Y -28.575,Z -41.130,A -90.000,B 90.000,C 0.000} C_DIS
LIN {X -103.375,Y -28.575,Z -40.519,A -90.000,B 90.000,C 0.000} C_DIS
LIN {X -102.754,Y -28.575,Z -39.951,A -90.000,B 90.000,C 0.000} C_DIS
LIN {X -102.094,Y -28.575,Z -39.429,A -90.000,B 90.000,C 0.000} C_DIS
LIN {X -101.986,Y -28.575,Z -39.330,A -90.000,B 90.000,C 0.000} C_DIS
LIN {X -101.353,Y -28.575,Z -38.853,A -90.000,B 90.000,C 0.000} C_DIS
LIN {X -100.687,Y -28.575,Z -38.422,A -90.000,B 90.000,C 0.000} C_DIS
LIN {X -99.993,Y -28.575,Z -38.040,A -90.000,B 90.000,C 0.000} C_DIS
LIN {X -99.273,Y -28.575,Z -37.709,A -90.000,B 90.000,C 0.000} C_DIS
LIN {X -98.321,Y -28.575,Z -37.368,A -90.000,B 90.000,C 0.000} C_DIS
LIN {X -97.351,Y -28.575,Z -37.082,A -90.000,B 90.000,C 0.000} C_DIS
LIN {X -96.366,Y -28.575,Z -36.852,A -90.000,B 90.000,C 0.000} C_DIS
LIN {X -95.370,Y -28.575,Z -36.680,A -90.000,B 90.000,C 0.000} C_DIS
LIN {X -94.365,Y -28.575,Z -36.565,A -90.000,B 90.000,C 0.000} C_DIS
LIN {X -93.355,Y -28.575,Z -36.508,A -90.000,B 90.000,C 0.000} C_DIS
LIN {X -92.344,Y -28.575,Z -36.509,A -90.000,B 90.000,C 0.000} C_DIS
LIN {X -91.334,Y -28.575,Z -36.569,A -90.000,B 90.000,C 0.000} C_DIS
LIN {X -90.330,Y -28.575,Z -36.686,A -90.000,B 90.000,C 0.000} C_DIS
LIN {X -89.790,Y -28.575,Z -36.024,A -90.000,B 90.000,C 0.000} C_DIS
LIN {X -89.209,Y -28.575,Z -35.397,A -90.000,B 90.000,C 0.000} C_DIS
LIN {X -88.589,Y -28.575,Z -34.809,A -90.000,B 90.000,C 0.000} C_DIS
LIN {X -87.933,Y -28.575,Z -34.262,A -90.000,B 90.000,C 0.000} C_DIS
LIN {X -87.243,Y -28.575,Z -33.758,A -90.000,B 90.000,C 0.000} C_DIS
LIN {X -86.523,Y -28.575,Z -33.299,A -90.000,B 90.000,C 0.000} C_DIS
LIN {X -85.774,Y -28.575,Z -32.887,A -90.000,B 90.000,C 0.000} C_DIS
LIN {X -85.001,Y -28.575,Z -32.524,A -90.000,B 90.000,C 0.000} C_DIS
LIN {X -84.049,Y -28.575,Z -32.225,A -90.000,B 90.000,C 0.000} C_DIS
LIN {X -83.080,Y -28.575,Z -31.985,A -90.000,B 90.000,C 0.000} C_DIS
LIN {X -82.099,Y -28.575,Z -31.805,A -90.000,B 90.000,C 0.000} C_DIS
LIN {X -81.108,Y -28.575,Z -31.686,A -90.000,B 90.000,C 0.000} C_DIS
LIN {X -80.111,Y -28.575,Z -31.629,A -90.000,B 90.000,C 0.000} C_DIS
LIN {X -79.114,Y -28.575,Z -31.633,A -90.000,B 90.000,C 0.000} C_DIS
LIN {X -78.118,Y -28.575,Z -31.699,A -90.000,B 90.000,C 0.000} C_DIS
LIN {X -77.128,Y -28.575,Z -31.827,A -90.000,B 90.000,C 0.000} C_DIS
LIN {X -75.467,Y -28.575,Z -32.172,A -90.000,B 90.000,C 0.000} C_DIS
LIN {X -73.817,Y -28.575,Z -32.566,A -90.000,B 90.000,C 0.000} C_DIS
LIN {X -72.179,Y -28.575,Z -33.008,A -90.000,B 90.000,C 0.000} C_DIS
LIN {X -70.554,Y -28.575,Z -33.498,A -90.000,B 90.000,C 0.000} C_DIS
LIN {X -68.945,Y -28.575,Z -34.035,A -90.000,B 90.000,C 0.000} C_DIS
LIN {X -67.352,Y -28.575,Z -34.619,A -90.000,B 90.000,C 0.000} C_DIS
LIN {X -65.777,Y -28.575,Z -35.250,A -90.000,B 90.000,C 0.000} C_DIS
LIN {X -64.135,Y -28.575,Z -36.034,A -90.000,B 90.000,C 0.000} C_DIS
LIN {X -62.475,Y -28.575,Z -36.776,A -90.000,B 90.000,C 0.000} C_DIS
LIN {X -60.795,Y -28.575,Z -37.475,A -90.000,B 90.000,C 0.000} C_DIS
LIN {X -59.099,Y -28.575,Z -38.131,A -90.000,B 90.000,C 0.000} C_DIS
LIN {X -57.386,Y -28.575,Z -38.744,A -90.000,B 90.000,C 0.000} C_DIS
LIN {X 21.387,Y -28.575,Z -38.744,A -90.000,B 90.000,C 0.000} C_DIS
LIN {X 22.487,Y -28.575,Z -38.266,A -90.000,B 90.000,C 0.000} C_DIS
LIN {X 23.606,Y -28.575,Z -37.833,A -90.000,B 90.000,C 0.000} C_DIS
LIN {X 24.741,Y -28.575,Z -37.446,A -90.000,B 90.000,C 0.000} C_DIS
LIN {X 25.891,Y -28.575,Z -37.105,A -90.000,B 90.000,C 0.000} C_DIS
LIN {X 27.053,Y -28.575,Z -36.811,A -90.000,B 90.000,C 0.000} C_DIS
LIN {X 28.227,Y -28.575,Z -36.564,A -90.000,B 90.000,C 0.000} C_DIS
LIN {X 29.111,Y -28.575,Z -36.474,A -90.000,B 90.000,C 0.000} C_DIS
LIN {X 29.987,Y -28.575,Z -36.330,A -90.000,B 90.000,C 0.000} C_DIS
LIN {X 30.853,Y -28.575,Z -36.132,A -90.000,B 90.000,C 0.000} C_DIS
LIN {X 31.705,Y -28.575,Z -35.880,A -90.000,B 90.000,C 0.000} C_DIS
LIN {X 32.540,Y -28.575,Z -35.577,A -90.000,B 90.000,C 0.000} C_DIS
LIN {X 33.768,Y -28.575,Z -35.076,A -90.000,B 90.000,C 0.000} C_DIS
LIN {X 35.016,Y -28.575,Z -34.629,A -90.000,B 90.000,C 0.000} C_DIS
LIN {X 36.283,Y -28.575,Z -34.239,A -90.000,B 90.000,C 0.000} C_DIS
LIN {X 37.567,Y -28.575,Z -33.904,A -90.000,B 90.000,C 0.000} C_DIS
LIN {X 38.863,Y -28.575,Z -33.626,A -90.000,B 90.000,C 0.000} C_DIS
LIN {X 40.171,Y -28.575,Z -33.406,A -90.000,B 90.000,C 0.000} C_DIS
LIN {X 41.487,Y -28.575,Z -33.244,A -90.000,B 90.000,C 0.000} C_DIS
LIN {X 42.809,Y -28.575,Z -33.140,A -90.000,B 90.000,C 0.000} C_DIS
LIN {X 44.141,Y -28.575,Z -33.165,A -90.000,B 90.000,C 0.000} C_DIS
LIN {X 45.470,Y -28.575,Z -33.252,A -90.000,B 90.000,C 0.000} C_DIS
LIN {X 46.793,Y -28.575,Z -33.400,A -90.000,B 90.000,C 0.000} C_DIS
LIN {X 48.108,Y -28.575,Z -33.609,A -90.000,B 90.000,C 0.000} C_DIS
LIN {X 49.413,Y -28.575,Z -33.879,A -90.000,B 90.000,C 0.000} C_DIS
LIN {X 50.703,Y -28.575,Z -34.209,A -90.000,B 90.000,C 0.000} C_DIS
LIN {X 51.977,Y -28.575,Z -34.598,A -90.000,B 90.000,C 0.000} C_DIS
LIN {X 53.231,Y -28.575,Z -35.045,A -90.000,B 90.000,C 0.000} C_DIS
LIN {X 54.606,Y -28.575,Z -35.696,A -90.000,B 90.000,C 0.000} C_DIS
LIN {X 55.958,Y -28.575,Z -36.392,A -90.000,B 90.000,C 0.000} C_DIS
LIN {X 57.287,Y -28.575,Z -37.133,A -90.000,B 90.000,C 0.000} C_DIS
LIN {X 58.590,Y -28.575,Z -37.917,A -90.000,B 90.000,C 0.000} C_DIS
LIN {X 59.867,Y -28.575,Z -38.744,A -90.000,B 90.000,C 0.000} C_DIS
LIN {X 85.657,Y -28.575,Z -38.744,A -90.000,B 90.000,C 0.000} C_DIS
LIN {X 84.505,Y -28.575,Z -39.705,A -90.000,B 90.000,C 0.000} C_DIS
LIN {X 83.389,Y -28.575,Z -40.707,A -90.000,B 90.000,C 0.000} C_DIS
LIN {X 82.311,Y -28.575,Z -41.749,A -90.000,B 90.000,C 0.000} C_DIS
LIN {X 81.271,Y -28.575,Z -42.831,A -90.000,B 90.000,C 0.000} C_DIS
LIN {X 80.272,Y -28.575,Z -43.950,A -90.000,B 90.000,C 0.000} C_DIS
LIN {X 79.315,Y -28.575,Z -45.104,A -90.000,B 90.000,C 0.000} C_DIS
LIN {X 78.400,Y -28.575,Z -46.293,A -90.000,B 90.000,C 0.000} C_DIS
LIN {X 68.670,Y -28.575,Z -46.293,A -90.000,B 90.000,C 0.000} C_DIS
LIN {X 70.523,Y -28.575,Z -48.925,A -90.000,B 90.000,C 0.000} C_DIS
LIN {X 71.915,Y -28.575,Z -49.738,A -90.000,B 90.000,C 0.000} C_DIS
LIN {X 73.284,Y -28.575,Z -50.587,A -90.000,B 90.000,C 0.000} C_DIS
LIN {X 74.632,Y -28.575,Z -51.472,A -90.000,B 90.000,C 0.000} C_DIS
LIN {X 75.955,Y -28.575,Z -52.392,A -90.000,B 90.000,C 0.000} C_DIS
LIN {X 76.430,Y -28.575,Z -51.380,A -90.000,B 90.000,C 0.000} C_DIS
LIN {X 76.940,Y -28.575,Z -50.385,A -90.000,B 90.000,C 0.000} C_DIS
LIN {X 77.484,Y -28.575,Z -49.408,A -90.000,B 90.000,C 0.000} C_DIS
LIN {X 78.417,Y -28.575,Z -47.991,A -90.000,B 90.000,C 0.000} C_DIS
LIN {X 79.409,Y -28.575,Z -46.615,A -90.000,B 90.000,C 0.000} C_DIS
LIN {X 80.458,Y -28.575,Z -45.282,A -90.000,B 90.000,C 0.000} C_DIS
LIN {X 81.563,Y -28.575,Z -43.995,A -90.000,B 90.000,C 0.000} C_DIS
LIN {X 82.722,Y -28.575,Z -42.757,A -90.000,B 90.000,C 0.000} C_DIS
LIN {X 83.933,Y -28.575,Z -41.568,A -90.000,B 90.000,C 0.000} C_DIS
LIN {X 85.193,Y -28.575,Z -40.433,A -90.000,B 90.000,C 0.000} C_DIS
LIN {X 86.500,Y -28.575,Z -39.351,A -90.000,B 90.000,C 0.000} C_DIS
LIN {X 87.852,Y -28.575,Z -38.327,A -90.000,B 90.000,C 0.000} C_DIS
LIN {X 89.246,Y -28.575,Z -37.360,A -90.000,B 90.000,C 0.000} C_DIS
LIN {X 91.067,Y -28.575,Z -36.216,A -90.000,B 90.000,C 0.000} C_DIS
LIN {X 92.918,Y -28.575,Z -35.121,A -90.000,B 90.000,C 0.000} C_DIS
LIN {X 94.797,Y -28.575,Z -34.076,A -90.000,B 90.000,C 0.000} C_DIS
LIN {X 96.704,Y -28.575,Z -33.081,A -90.000,B 90.000,C 0.000} C_DIS
LIN {X 98.636,Y -28.575,Z -32.137,A -90.000,B 90.000,C 0.000} C_DIS
LIN {X 100.592,Y -28.575,Z -31.245,A -90.000,B 90.000,C 0.000} C_DIS
LIN {X 102.572,Y -28.575,Z -30.405,A -90.000,B 90.000,C 0.000} C_DIS
LIN {X 104.573,Y -28.575,Z -29.618,A -90.000,B 90.000,C 0.000} C_DIS
LIN {X 105.513,Y -28.575,Z -29.233,A -90.000,B 90.000,C 0.000} C_DIS
LIN {X 106.478,Y -28.575,Z -28.915,A -90.000,B 90.000,C 0.000} C_DIS
LIN {X 107.464,Y -28.575,Z -28.667,A -90.000,B 90.000,C 0.000} C_DIS
LIN {X 108.464,Y -28.575,Z -28.489,A -90.000,B 90.000,C 0.000} C_DIS
LIN {X 109.474,Y -28.575,Z -28.382,A -90.000,B 90.000,C 0.000} C_DIS
LIN {X 110.490,Y -28.575,Z -28.346,A -90.000,B 90.000,C 0.000} C_DIS
LIN {X 111.505,Y -28.575,Z -28.383,A -90.000,B 90.000,C 0.000} C_DIS
LIN {X 112.516,Y -28.575,Z -28.492,A -90.000,B 90.000,C 0.000} C_DIS
LIN {X 113.516,Y -28.575,Z -28.671,A -90.000,B 90.000,C 0.000} C_DIS
LIN {X 114.501,Y -28.575,Z -28.921,A -90.000,B 90.000,C 0.000} C_DIS
LIN {X 115.465,Y -28.575,Z -29.240,A -90.000,B 90.000,C 0.000} C_DIS
LIN {X 116.405,Y -28.575,Z -29.627,A -90.000,B 90.000,C 0.000} C_DIS
LIN {X 117.315,Y -28.575,Z -30.079,A -90.000,B 90.000,C 0.000} C_DIS
LIN {X 118.191,Y -28.575,Z -30.594,A -90.000,B 90.000,C 0.000} C_DIS
LIN {X 119.028,Y -28.575,Z -31.170,A -90.000,B 90.000,C 0.000} C_DIS
LIN {X 119.134,Y -28.575,Z -31.254,A -90.000,B 90.000,C 0.000} C_DIS
LIN {X 119.817,Y -28.575,Z -31.832,A -90.000,B 90.000,C 0.000} C_DIS
LIN {X 120.468,Y -28.575,Z -32.447,A -90.000,B 90.000,C 0.000} C_DIS
LIN {X 121.083,Y -28.575,Z -33.097,A -90.000,B 90.000,C 0.000} C_DIS
LIN {X 121.662,Y -28.575,Z -33.780,A -90.000,B 90.000,C 0.000} C_DIS
LIN {X 122.196,Y -28.575,Z -34.612,A -90.000,B 90.000,C 0.000} C_DIS
LIN {X 122.676,Y -28.575,Z -35.476,A -90.000,B 90.000,C 0.000} C_DIS
LIN {X 123.102,Y -28.575,Z -36.368,A -90.000,B 90.000,C 0.000} C_DIS
LIN {X 123.470,Y -28.575,Z -37.286,A -90.000,B 90.000,C 0.000} C_DIS
LIN {X 123.781,Y -28.575,Z -38.224,A -90.000,B 90.000,C 0.000} C_DIS
LIN {X 124.032,Y -28.575,Z -39.180,A -90.000,B 90.000,C 0.000} C_DIS
LIN {X 124.222,Y -28.575,Z -40.150,A -90.000,B 90.000,C 0.000} C_DIS
LIN {X 124.352,Y -28.575,Z -41.130,A -90.000,B 90.000,C 0.000} C_DIS
LIN {X 124.419,Y -28.575,Z -42.117,A -90.000,B 90.000,C 0.000} C_DIS
LIN {X 124.425,Y -28.575,Z -43.105,A -90.000,B 90.000,C 0.000} C_DIS
LIN {X 124.369,Y -28.575,Z -44.092,A -90.000,B 90.000,C 0.000} C_DIS
LIN {X 124.170,Y -28.575,Z -45.366,A -90.000,B 90.000,C 0.000} C_DIS
LIN {X 123.911,Y -28.575,Z -46.630,A -90.000,B 90.000,C 0.000} C_DIS
LIN {X 123.595,Y -28.575,Z -47.880,A -90.000,B 90.000,C 0.000} C_DIS
LIN {X 123.220,Y -28.575,Z -49.114,A -90.000,B 90.000,C 0.000} C_DIS
LIN {X 122.789,Y -28.575,Z -50.330,A -90.000,B 90.000,C 0.000} C_DIS
LIN {X 122.302,Y -28.575,Z -51.524,A -90.000,B 90.000,C 0.000} C_DIS
LIN {X 121.760,Y -28.575,Z -52.694,A -90.000,B 90.000,C 0.000} C_DIS
LIN {X 121.061,Y -28.575,Z -53.939,A -90.000,B 90.000,C 0.000} C_DIS
LIN {X 120.409,Y -28.575,Z -55.208,A -90.000,B 90.000,C 0.000} C_DIS
LIN {X 119.804,Y -28.575,Z -56.501,A -90.000,B 90.000,C 0.000} C_DIS
LIN {X 119.247,Y -28.575,Z -57.815,A -90.000,B 90.000,C 0.000} C_DIS
LIN {X 118.739,Y -28.575,Z -59.149,A -90.000,B 90.000,C 0.000} C_DIS
LIN {X 118.281,Y -28.575,Z -60.500,A -90.000,B 90.000,C 0.000} C_DIS
LIN {X 117.872,Y -28.575,Z -61.868,A -90.000,B 90.000,C 0.000} C_DIS
LIN {X 117.358,Y -28.575,Z -63.979,A -90.000,B 90.000,C 0.000} C_DIS
LIN {X 116.784,Y -28.575,Z -66.075,A -90.000,B 90.000,C 0.000} C_DIS
LIN {X 116.150,Y -28.575,Z -68.153,A -90.000,B 90.000,C 0.000} C_DIS
LIN {X 115.456,Y -28.575,Z -70.212,A -90.000,B 90.000,C 0.000} C_DIS
LIN {X 114.703,Y -28.575,Z -72.250,A -90.000,B 90.000,C 0.000} C_DIS
LIN {X 113.892,Y -28.575,Z -74.265,A -90.000,B 90.000,C 0.000} C_DIS
LIN {X 113.023,Y -28.575,Z -76.257,A -90.000,B 90.000,C 0.000} C_DIS
LIN {X 112.096,Y -28.575,Z -78.222,A -90.000,B 90.000,C 0.000} C_DIS
LIN {X 111.114,Y -28.575,Z -80.160,A -90.000,B 90.000,C 0.000} C_DIS
LIN {X 110.076,Y -28.575,Z -82.069,A -90.000,B 90.000,C 0.000} C_DIS
LIN {X 108.984,Y -28.575,Z -83.947,A -90.000,B 90.000,C 0.000} C_DIS
LIN {X 107.838,Y -28.575,Z -85.793,A -90.000,B 90.000,C 0.000} C_DIS
LIN {X 106.639,Y -28.575,Z -87.605,A -90.000,B 90.000,C 0.000} C_DIS
LIN {X 106.770,Y -28.575,Z -89.236,A -90.000,B 90.000,C 0.000} C_DIS
LIN {X 106.855,Y -28.575,Z -90.869,A -90.000,B 90.000,C 0.000} C_DIS
LIN {X 106.892,Y -28.575,Z -92.505,A -90.000,B 90.000,C 0.000} C_DIS
LIN {X 106.883,Y -28.575,Z -94.140,A -90.000,B 90.000,C 0.000} C_DIS
LIN {X 106.827,Y -28.575,Z -95.775,A -90.000,B 90.000,C 0.000} C_DIS
LIN {X 106.725,Y -28.575,Z -97.408,A -90.000,B 90.000,C 0.000} C_DIS
LIN {X 106.726,Y -28.575,Z -97.579,A -90.000,B 90.000,C 0.000} C_DIS
LIN {X 106.611,Y -28.575,Z -99.046,A -90.000,B 90.000,C 0.000} C_DIS
LIN {X 106.530,Y -28.575,Z -100.516,A -90.000,B 90.000,C 0.000} C_DIS
LIN {X 106.484,Y -28.575,Z -101.986,A -90.000,B 90.000,C 0.000} C_DIS
LIN {X 106.472,Y -28.575,Z -103.458,A -90.000,B 90.000,C 0.000} C_DIS
LIN {X 106.719,Y -28.575,Z -104.871,A -90.000,B 90.000,C 0.000} C_DIS
LIN {X 106.922,Y -28.575,Z -106.292,A -90.000,B 90.000,C 0.000} C_DIS
LIN {X 107.081,Y -28.575,Z -107.718,A -90.000,B 90.000,C 0.000} C_DIS
LIN {X 107.195,Y -28.575,Z -109.148,A -90.000,B 90.000,C 0.000} C_DIS
LIN {X 107.496,Y -28.575,Z -112.271,A -90.000,B 90.000,C 0.000} C_DIS
LIN {X 107.744,Y -28.575,Z -115.399,A -90.000,B 90.000,C 0.000} C_DIS
LIN {X 107.940,Y -28.575,Z -118.530,A -90.000,B 90.000,C 0.000} C_DIS
LIN {X 108.084,Y -28.575,Z -121.665,A -90.000,B 90.000,C 0.000} C_DIS
LIN {X 108.176,Y -28.575,Z -124.801,A -90.000,B 90.000,C 0.000} C_DIS
LIN {X 108.062,Y -28.575,Z -129.028,A -90.000,B 90.000,C 0.000} C_DIS
LIN {X 107.892,Y -28.575,Z -133.253,A -90.000,B 90.000,C 0.000} C_DIS
LIN {X 107.668,Y -28.575,Z -137.475,A -90.000,B 90.000,C 0.000} C_DIS
LIN {X 107.388,Y -28.575,Z -141.694,A -90.000,B 90.000,C 0.000} C_DIS
LIN {X 107.053,Y -28.575,Z -145.910,A -90.000,B 90.000,C 0.000} C_DIS
LIN {X 106.664,Y -28.575,Z -150.120,A -90.000,B 90.000,C 0.000} C_DIS
LIN {X 106.236,Y -28.575,Z -153.765,A -90.000,B 90.000,C 0.000} C_DIS
LIN {X 105.831,Y -28.575,Z -157.412,A -90.000,B 90.000,C 0.000} C_DIS
LIN {X 105.396,Y -28.575,Z -160.199,A -90.000,B 90.000,C 0.000} C_DIS
LIN {X 104.998,Y -28.575,Z -162.993,A -90.000,B 90.000,C 0.000} C_DIS
LIN {X 104.639,Y -28.575,Z -165.791,A -90.000,B 90.000,C 0.000} C_DIS
LIN {X 104.318,Y -28.575,Z -168.594,A -90.000,B 90.000,C 0.000} C_DIS
LIN {X 103.865,Y -28.575,Z -171.249,A -90.000,B 90.000,C 0.000} C_DIS
LIN {X 103.458,Y -28.575,Z -173.913,A -90.000,B 90.000,C 0.000} C_DIS
LIN {X 103.099,Y -28.575,Z -176.582,A -90.000,B 90.000,C 0.000} C_DIS
LIN {X 102.786,Y -28.575,Z -179.258,A -90.000,B 90.000,C 0.000} C_DIS
LIN {X 102.522,Y -28.575,Z -181.939,A -90.000,B 90.000,C 0.000} C_DIS
LIN {X 102.304,Y -28.575,Z -184.624,A -90.000,B 90.000,C 0.000} C_DIS
LIN {X 102.170,Y -28.575,Z -187.191,A -90.000,B 90.000,C 0.000} C_DIS
LIN {X 101.988,Y -28.575,Z -189.756,A -90.000,B 90.000,C 0.000} C_DIS
LIN {X 101.759,Y -28.575,Z -192.317,A -90.000,B 90.000,C 0.000} C_DIS
LIN {X 101.483,Y -28.575,Z -194.873,A -90.000,B 90.000,C 0.000} C_DIS
LIN {X 101.160,Y -28.575,Z -197.423,A -90.000,B 90.000,C 0.000} C_DIS
LIN {X 100.468,Y -28.575,Z -200.948,A -90.000,B 90.000,C 0.000} C_DIS
LIN {X 99.719,Y -28.575,Z -204.462,A -90.000,B 90.000,C 0.000} C_DIS
LIN {X 98.913,Y -28.575,Z -207.963,A -90.000,B 90.000,C 0.000} C_DIS
LIN {X 98.051,Y -28.575,Z -211.451,A -90.000,B 90.000,C 0.000} C_DIS
LIN {X 97.133,Y -28.575,Z -214.924,A -90.000,B 90.000,C 0.000} C_DIS
LIN {X 95.887,Y -28.575,Z -219.700,A -90.000,B 90.000,C 0.000} C_DIS
LIN {X 94.665,Y -28.575,Z -224.483,A -90.000,B 90.000,C 0.000} C_DIS
LIN {X 93.889,Y -28.575,Z -227.699,A -90.000,B 90.000,C 0.000} C_DIS
LIN {X 93.060,Y -28.575,Z -230.901,A -90.000,B 90.000,C 0.000} C_DIS
LIN {X 92.178,Y -28.575,Z -234.089,A -90.000,B 90.000,C 0.000} C_DIS
LIN {X 91.243,Y -28.575,Z -237.263,A -90.000,B 90.000,C 0.000} C_DIS
LIN {X 90.257,Y -28.575,Z -240.420,A -90.000,B 90.000,C 0.000} C_DIS
LIN {X 89.218,Y -28.575,Z -243.561,A -90.000,B 90.000,C 0.000} C_DIS
LIN {X 145.015,Y -28.575,Z -243.561,A -90.000,B 90.000,C 0.000} C_DIS
LIN {X 145.015,Y -28.575,Z 0.000,A -90.000,B 90.000,C 0.000} C_DIS
LIN {X -145.015,Y -28.575,Z 0.000,A -90.000,B 90.000,C 0.000} C_DIS
LIN {X -145.015,Y -28.575,Z -243.561,A -90.000,B 90.000,C 0.000} C_DIS
LIN {X -117.147,Y -28.575,Z -243.561,A -90.000,B 90.000,C 0.000} C_DIS
LIN {X -112.160,Y -28.575,Z -240.051,A -90.000,B 90.000,C 0.000} C_DIS
LIN {X -107.140,Y -28.575,Z -236.590,A -90.000,B 90.000,C 0.000} C_DIS
LIN {X -102.085,Y -28.575,Z -233.179,A -90.000,B 90.000,C 0.000} C_DIS
LIN {X -96.998,Y -28.575,Z -229.817,A -90.000,B 90.000,C 0.000} C_DIS
LIN {X -91.877,Y -28.575,Z -226.505,A -90.000,B 90.000,C 0.000} C_DIS
LIN {X -86.724,Y -28.575,Z -223.244,A -90.000,B 90.000,C 0.000} C_DIS
LIN {X -81.540,Y -28.575,Z -220.034,A -90.000,B 90.000,C 0.000} C_DIS
LIN {X -76.324,Y -28.575,Z -216.874,A -90.000,B 90.000,C 0.000} C_DIS
LIN {X -71.078,Y -28.575,Z -213.766,A -90.000,B 90.000,C 0.000} C_DIS
LIN {X -63.645,Y -28.575,Z -209.440,A -90.000,B 90.000,C 0.000} C_DIS
LIN {X -56.401,Y -28.575,Z -205.291,A -90.000,B 90.000,C 0.000} C_DIS
LIN {X -50.769,Y -28.575,Z -202.092,A -90.000,B 90.000,C 0.000} C_DIS
LIN {X -45.163,Y -28.575,Z -198.848,A -90.000,B 90.000,C 0.000} C_DIS
LIN {X -39.583,Y -28.575,Z -195.559,A -90.000,B 90.000,C 0.000} C_DIS
LIN {X -37.656,Y -28.575,Z -194.467,A -90.000,B 90.000,C 0.000} C_DIS
LIN {X -35.762,Y -28.575,Z -193.317,A -90.000,B 90.000,C 0.000} C_DIS
LIN {X -33.904,Y -28.575,Z -192.111,A -90.000,B 90.000,C 0.000} C_DIS
LIN {X -32.084,Y -28.575,Z -190.850,A -90.000,B 90.000,C 0.000} C_DIS
LIN {X -30.302,Y -28.575,Z -189.534,A -90.000,B 90.000,C 0.000} C_DIS
LIN {X -28.561,Y -28.575,Z -188.165,A -90.000,B 90.000,C 0.000} C_DIS
LIN {X -26.861,Y -28.575,Z -186.744,A -90.000,B 90.000,C 0.000} C_DIS
LIN {X -25.206,Y -28.575,Z -185.272,A -90.000,B 90.000,C 0.000} C_DIS
LIN {X -23.595,Y -28.575,Z -183.752,A -90.000,B 90.000,C 0.000} C_DIS
LIN {X -22.031,Y -28.575,Z -182.183,A -90.000,B 90.000,C 0.000} C_DIS
LIN {X -20.738,Y -28.575,Z -180.898,A -90.000,B 90.000,C 0.000} C_DIS
LIN {X -19.493,Y -28.575,Z -179.568,A -90.000,B 90.000,C 0.000} C_DIS
LIN {X -18.296,Y -28.575,Z -178.193,A -90.000,B 90.000,C 0.000} C_DIS
LIN {X -17.149,Y -28.575,Z -176.777,A -90.000,B 90.000,C 0.000} C_DIS
LIN {X -16.053,Y -28.575,Z -175.321,A -90.000,B 90.000,C 0.000} C_DIS
LIN {X -15.010,Y -28.575,Z -173.826,A -90.000,B 90.000,C 0.000} C_DIS
LIN {X -14.022,Y -28.575,Z -172.295,A -90.000,B 90.000,C 0.000} C_DIS
LIN {X -13.089,Y -28.575,Z -170.729,A -90.000,B 90.000,C 0.000} C_DIS
LIN {X -12.624,Y -28.575,Z -169.926,A -90.000,B 90.000,C 0.000} C_DIS
LIN {X -12.209,Y -28.575,Z -169.096,A -90.000,B 90.000,C 0.000} C_DIS
LIN {X -11.845,Y -28.575,Z -168.241,A -90.000,B 90.000,C 0.000} C_DIS
LIN {X -11.535,Y -28.575,Z -167.367,A -90.000,B 90.000,C 0.000} C_DIS
LIN {X -11.279,Y -28.575,Z -166.474,A -90.000,B 90.000,C 0.000} C_DIS
LIN {X -11.079,Y -28.575,Z -165.568,A -90.000,B 90.000,C 0.000} C_DIS
LIN {X -10.935,Y -28.575,Z -164.651,A -90.000,B 90.000,C 0.000} C_DIS
LIN {X -12.681,Y -28.575,Z -163.239,A -90.000,B 90.000,C 0.000} C_DIS
LIN {X -14.451,Y -28.575,Z -161.858,A -90.000,B 90.000,C 0.000} C_DIS
LIN {X -16.787,Y -28.575,Z -160.106,A -90.000,B 90.000,C 0.000} C_DIS
LIN {X -19.089,Y -28.575,Z -158.308,A -90.000,B 90.000,C 0.000} C_DIS
LIN {X -21.356,Y -28.575,Z -156.467,A -90.000,B 90.000,C 0.000} C_DIS
LIN {X -23.587,Y -28.575,Z -154.583,A -90.000,B 90.000,C 0.000} C_DIS
LIN {X -25.781,Y -28.575,Z -152.656,A -90.000,B 90.000,C 0.000} C_DIS
LIN {X -27.938,Y -28.575,Z -150.687,A -90.000,B 90.000,C 0.000} C_DIS
LIN {X -29.220,Y -28.575,Z -149.483,A -90.000,B 90.000,C 0.000} C_DIS
LIN {X -30.464,Y -28.575,Z -148.240,A -90.000,B 90.000,C 0.000} C_DIS
LIN {X -31.669,Y -28.575,Z -146.959,A -90.000,B 90.000,C 0.000} C_DIS
LIN {X -32.834,Y -28.575,Z -145.642,A -90.000,B 90.000,C 0.000} C_DIS
LIN {X -33.958,Y -28.575,Z -144.290,A -90.000,B 90.000,C 0.000} C_DIS
LIN {X -35.040,Y -28.575,Z -142.904,A -90.000,B 90.000,C 0.000} C_DIS
LIN {X -36.079,Y -28.575,Z -141.485,A -90.000,B 90.000,C 0.000} C_DIS
LIN {X -37.438,Y -28.575,Z -139.749,A -90.000,B 90.000,C 0.000} C_DIS
LIN {X -38.746,Y -28.575,Z -137.974,A -90.000,B 90.000,C 0.000} C_DIS
LIN {X -40.000,Y -28.575,Z -136.161,A -90.000,B 90.000,C 0.000} C_DIS
LIN {X -41.200,Y -28.575,Z -134.312,A -90.000,B 90.000,C 0.000} C_DIS
LIN {X -42.344,Y -28.575,Z -132.427,A -90.000,B 90.000,C 0.000} C_DIS
LIN {X -43.433,Y -28.575,Z -130.510,A -90.000,B 90.000,C 0.000} C_DIS
LIN {X -44.463,Y -28.575,Z -128.561,A -90.000,B 90.000,C 0.000} C_DIS
LIN {X -45.843,Y -28.575,Z -125.543,A -90.000,B 90.000,C 0.000} C_DIS
LIN {X -47.246,Y -28.575,Z -122.534,A -90.000,B 90.000,C 0.000} C_DIS
LIN {X -48.671,Y -28.575,Z -119.537,A -90.000,B 90.000,C 0.000} C_DIS
LIN {X -49.913,Y -28.575,Z -117.548,A -90.000,B 90.000,C 0.000} C_DIS
LIN {X -51.200,Y -28.575,Z -115.586,A -90.000,B 90.000,C 0.000} C_DIS
LIN {X -52.530,Y -28.575,Z -113.654,A -90.000,B 90.000,C 0.000} C_DIS
LIN {X -53.902,Y -28.575,Z -111.752,A -90.000,B 90.000,C 0.000} C_DIS
LIN {X -55.316,Y -28.575,Z -109.881,A -90.000,B 90.000,C 0.000} C_DIS
LIN {X -56.772,Y -28.575,Z -108.042,A -90.000,B 90.000,C 0.000} C_DIS
LIN {X -58.562,Y -28.575,Z -105.754,A -90.000,B 90.000,C 0.000} C_DIS
LIN {X -60.324,Y -28.575,Z -103.445,A -90.000,B 90.000,C 0.000} C_DIS
LIN {X -61.865,Y -28.575,Z -101.283,A -90.000,B 90.000,C 0.000} C_DIS
LIN {X -63.445,Y -28.575,Z -99.150,A -90.000,B 90.000,C 0.000} C_DIS
LIN {X -65.065,Y -28.575,Z -97.048,A -90.000,B 90.000,C 0.000} C_DIS
LIN {X -66.724,Y -28.575,Z -94.975,A -90.000,B 90.000,C 0.000} C_DIS
LIN {X -68.421,Y -28.575,Z -92.934,A -90.000,B 90.000,C 0.000} C_DIS
LIN {X -70.156,Y -28.575,Z -90.925,A -90.000,B 90.000,C 0.000} C_DIS
LIN {X -71.862,Y -28.575,Z -89.106,A -90.000,B 90.000,C 0.000} C_DIS
LIN {X -73.550,Y -28.575,Z -87.270,A -90.000,B 90.000,C 0.000} C_DIS
LIN {X -75.852,Y -28.575,Z -84.818,A -90.000,B 90.000,C 0.000} C_DIS
LIN {X -78.144,Y -28.575,Z -82.356,A -90.000,B 90.000,C 0.000} C_DIS
LIN {X -79.209,Y -28.575,Z -82.203,A -90.000,B 90.000,C 0.000} C_DIS
LIN {X -80.261,Y -28.575,Z -81.982,A -90.000,B 90.000,C 0.000} C_DIS
LIN {X -81.298,Y -28.575,Z -81.694,A -90.000,B 90.000,C 0.000} C_DIS
LIN {X -82.313,Y -28.575,Z -81.339,A -90.000,B 90.000,C 0.000} C_DIS
LIN {X -83.304,Y -28.575,Z -80.920,A -90.000,B 90.000,C 0.000} C_DIS
LIN {X -84.265,Y -28.575,Z -80.438,A -90.000,B 90.000,C 0.000} C_DIS
LIN {X -85.194,Y -28.575,Z -79.896,A -90.000,B 90.000,C 0.000} C_DIS
LIN {X -86.086,Y -28.575,Z -79.294,A -90.000,B 90.000,C 0.000} C_DIS
LIN {X -86.937,Y -28.575,Z -78.637,A -90.000,B 90.000,C 0.000} C_DIS
LIN {X -87.744,Y -28.575,Z -77.926,A -90.000,B 90.000,C 0.000} C_DIS
LIN {X -88.504,Y -28.575,Z -77.165,A -90.000,B 90.000,C 0.000} C_DIS
LIN {X -89.214,Y -28.575,Z -76.357,A -90.000,B 90.000,C 0.000} C_DIS
LIN {X -89.870,Y -28.575,Z -75.504,A -90.000,B 90.000,C 0.000} C_DIS
LIN {X -90.470,Y -28.575,Z -74.611,A -90.000,B 90.000,C 0.000} C_DIS
LIN {X -91.011,Y -28.575,Z -73.682,A -90.000,B 90.000,C 0.000} C_DIS
LIN {X -91.387,Y -28.575,Z -72.988,A -90.000,B 90.000,C 0.000} C_DIS
LIN {X -91.715,Y -28.575,Z -72.270,A -90.000,B 90.000,C 0.000} C_DIS
LIN {X -91.993,Y -28.575,Z -71.532,A -90.000,B 90.000,C 0.000} C_DIS
LIN {X -92.221,Y -28.575,Z -70.776,A -90.000,B 90.000,C 0.000} C_DIS
LIN {X -92.397,Y -28.575,Z -70.007,A -90.000,B 90.000,C 0.000} C_DIS
LIN {X -92.519,Y -28.575,Z -69.227,A -90.000,B 90.000,C 0.000} C_DIS
LIN {X -93.180,Y -28.575,Z -68.691,A -90.000,B 90.000,C 0.000} C_DIS
LIN {X -93.828,Y -28.575,Z -68.140,A -90.000,B 90.000,C 0.000} C_DIS
LIN {X -94.463,Y -28.575,Z -67.574,A -90.000,B 90.000,C 0.000} C_DIS
LIN {X -94.602,Y -28.575,Z -67.443,A -90.000,B 90.000,C 0.000} C_DIS
LIN {X -95.164,Y -28.575,Z -66.865,A -90.000,B 90.000,C 0.000} C_DIS
LIN {X -95.686,Y -28.575,Z -66.252,A -90.000,B 90.000,C 0.000} C_DIS
LIN {X -96.166,Y -28.575,Z -65.605,A -90.000,B 90.000,C 0.000} C_DIS
LIN {X -96.602,Y -28.575,Z -64.928,A -90.000,B 90.000,C 0.000} C_DIS
LIN {X -96.992,Y -28.575,Z -64.223,A -90.000,B 90.000,C 0.000} C_DIS
LIN {X -97.335,Y -28.575,Z -63.494,A -90.000,B 90.000,C 0.000} C_DIS
LIN {X -98.348,Y -28.575,Z -62.616,A -90.000,B 90.000,C 0.000} C_DIS
LIN {X -99.335,Y -28.575,Z -61.709,A -90.000,B 90.000,C 0.000} C_DIS
LIN {X -100.295,Y -28.575,Z -60.773,A -90.000,B 90.000,C 0.000} C_DIS
LIN {X -101.228,Y -28.575,Z -59.810,A -90.000,B 90.000,C 0.000} C_DIS
LIN {X -102.132,Y -28.575,Z -58.820,A -90.000,B 90.000,C 0.000} C_DIS
LIN {X -102.256,Y -28.575,Z -58.674,A -90.000,B 90.000,C 0.000} C_DIS
LIN {X -102.758,Y -28.575,Z -58.043,A -90.000,B 90.000,C 0.000} C_DIS
LIN {X -103.227,Y -28.575,Z -57.386,A -90.000,B 90.000,C 0.000} C_DIS
LIN {X -103.661,Y -28.575,Z -56.705,A -90.000,B 90.000,C 0.000} C_DIS
LIN {X -104.058,Y -28.575,Z -56.003,A -90.000,B 90.000,C 0.000} C_DIS
LIN {X -104.418,Y -28.575,Z -55.281,A -90.000,B 90.000,C 0.000} C_DIS
LIN {X -104.829,Y -28.575,Z -54.465,A -90.000,B 90.000,C 0.000} C_DIS
LIN {X -105.177,Y -28.575,Z -53.620,A -90.000,B 90.000,C 0.000} C_DIS
LIN {X -105.460,Y -28.575,Z -52.752,A -90.000,B 90.000,C 0.000} C_DIS
LIN {X -105.677,Y -28.575,Z -51.864,A -90.000,B 90.000,C 0.000} C_DIS
LIN {X -105.825,Y -28.575,Z -50.962,A -90.000,B 90.000,C 0.000} C_DIS
LIN {X -105.905,Y -28.575,Z -50.052,A -90.000,B 90.000,C 0.000} C_DIS
LIN {X -105.915,Y -28.575,Z -49.138,A -90.000,B 90.000,C 0.000} C_DIS
LIN {X -105.856,Y -28.575,Z -48.227,A -90.000,B 90.000,C 0.000} C_DIS
LIN {X -105.728,Y -28.575,Z -47.322,A -90.000,B 90.000,C 0.000} C_DIS
LIN {X -105.578,Y -28.575,Z -46.483,A -90.000,B 90.000,C 0.000} C_DIS
LIN {X -105.360,Y -28.575,Z -45.659,A -90.000,B 90.000,C 0.000} C_DIS
LIN {X -105.077,Y -28.575,Z -44.854,A -90.000,B 90.000,C 0.000} C_DIS
LIN {X -104.730,Y -28.575,Z -44.076,A -90.000,B 90.000,C 0.000} C_DIS
LIN {X -104.322,Y -28.575,Z -43.328,A -90.000,B 90.000,C 0.000} C_DIS
LIN {X -103.854,Y -28.575,Z -42.615,A -90.000,B 90.000,C 0.000} C_DIS
LIN {X -103.331,Y -28.575,Z -41.942,A -90.000,B 90.000,C 0.000} C_DIS
LIN {X -102.755,Y -28.575,Z -41.313,A -90.000,B 90.000,C 0.000} C_DIS
LIN {X -102.130,Y -28.575,Z -40.733,A -90.000,B 90.000,C 0.000} C_DIS
LIN {X -101.461,Y -28.575,Z -40.205,A -90.000,B 90.000,C 0.000} C_DIS
LIN {X -101.334,Y -28.575,Z -40.089,A -90.000,B 90.000,C 0.000} C_DIS
LIN {X -100.765,Y -28.575,Z -39.662,A -90.000,B 90.000,C 0.000} C_DIS
LIN {X -100.167,Y -28.575,Z -39.276,A -90.000,B 90.000,C 0.000} C_DIS
LIN {X -99.543,Y -28.575,Z -38.934,A -90.000,B 90.000,C 0.000} C_DIS
LIN {X -98.897,Y -28.575,Z -38.636,A -90.000,B 90.000,C 0.000} C_DIS
LIN {X -97.937,Y -28.575,Z -38.295,A -90.000,B 90.000,C 0.000} C_DIS
LIN {X -96.958,Y -28.575,Z -38.013,A -90.000,B 90.000,C 0.000} C_DIS
LIN {X -95.963,Y -28.575,Z -37.793,A -90.000,B 90.000,C 0.000} C_DIS
LIN {X -94.957,Y -28.575,Z -37.633,A -90.000,B 90.000,C 0.000} C_DIS
LIN {X -93.943,Y -28.575,Z -37.536,A -90.000,B 90.000,C 0.000} C_DIS
LIN {X -92.925,Y -28.575,Z -37.502,A -90.000,B 90.000,C 0.000} C_DIS
LIN {X -91.906,Y -28.575,Z -37.530,A -90.000,B 90.000,C 0.000} C_DIS
LIN {X -90.891,Y -28.575,Z -37.620,A -90.000,B 90.000,C 0.000} C_DIS
LIN {X -89.884,Y -28.575,Z -37.773,A -90.000,B 90.000,C 0.000} C_DIS
LIN {X -89.371,Y -28.575,Z -37.082,A -90.000,B 90.000,C 0.000} C_DIS
LIN {X -88.812,Y -28.575,Z -36.429,A -90.000,B 90.000,C 0.000} C_DIS
LIN {X -88.208,Y -28.575,Z -35.816,A -90.000,B 90.000,C 0.000} C_DIS
LIN {X -87.564,Y -28.575,Z -35.247,A -90.000,B 90.000,C 0.000} C_DIS
LIN {X -86.881,Y -28.575,Z -34.724,A -90.000,B 90.000,C 0.000} C_DIS
LIN {X -86.163,Y -28.575,Z -34.250,A -90.000,B 90.000,C 0.000} C_DIS
LIN {X -85.415,Y -28.575,Z -33.827,A -90.000,B 90.000,C 0.000} C_DIS
LIN {X -84.638,Y -28.575,Z -33.457,A -90.000,B 90.000,C 0.000} C_DIS
LIN {X -83.750,Y -28.575,Z -33.180,A -90.000,B 90.000,C 0.000} C_DIS
LIN {X -82.847,Y -28.575,Z -32.958,A -90.000,B 90.000,C 0.000} C_DIS
LIN {X -81.933,Y -28.575,Z -32.792,A -90.000,B 90.000,C 0.000} C_DIS
LIN {X -81.009,Y -28.575,Z -32.682,A -90.000,B 90.000,C 0.000} C_DIS
LIN {X -80.081,Y -28.575,Z -32.629,A -90.000,B 90.000,C 0.000} C_DIS
LIN {X -79.151,Y -28.575,Z -32.633,A -90.000,B 90.000,C 0.000} C_DIS
LIN {X -78.223,Y -28.575,Z -32.694,A -90.000,B 90.000,C 0.000} C_DIS
LIN {X -77.301,Y -28.575,Z -32.812,A -90.000,B 90.000,C 0.000} C_DIS
LIN {X -75.405,Y -28.575,Z -33.211,A -90.000,B 90.000,C 0.000} C_DIS
LIN {X -73.524,Y -28.575,Z -33.675,A -90.000,B 90.000,C 0.000} C_DIS
LIN {X -71.660,Y -28.575,Z -34.202,A -90.000,B 90.000,C 0.000} C_DIS
LIN {X -69.815,Y -28.575,Z -34.793,A -90.000,B 90.000,C 0.000} C_DIS
LIN {X -67.991,Y -28.575,Z -35.446,A -90.000,B 90.000,C 0.000} C_DIS
LIN {X -66.191,Y -28.575,Z -36.161,A -90.000,B 90.000,C 0.000} C_DIS
LIN {X -64.247,Y -28.575,Z -37.083,A -90.000,B 90.000,C 0.000} C_DIS
LIN {X -62.277,Y -28.575,Z -37.947,A -90.000,B 90.000,C 0.000} C_DIS
LIN {X -60.282,Y -28.575,Z -38.752,A -90.000,B 90.000,C 0.000} C_DIS
LIN {X -58.264,Y -28.575,Z -39.497,A -90.000,B 90.000,C 0.000} C_DIS
LIN {X -56.225,Y -28.575,Z -40.183,A -90.000,B 90.000,C 0.000} C_DIS
LIN {X -54.166,Y -28.575,Z -40.807,A -90.000,B 90.000,C 0.000} C_DIS
LIN {X -53.979,Y -28.575,Z -40.852,A -90.000,B 90.000,C 0.000} C_DIS
LIN {X -52.601,Y -28.575,Z -41.128,A -90.000,B 90.000,C 0.000} C_DIS
LIN {X -49.545,Y -28.575,Z -41.414,A -90.000,B 90.000,C 0.000} C_DIS
LIN {X -46.496,Y -28.575,Z -41.768,A -90.000,B 90.000,C 0.000} C_DIS
LIN {X -43.455,Y -28.575,Z -42.187,A -90.000,B 90.000,C 0.000} C_DIS
LIN {X -40.424,Y -28.575,Z -42.674,A -90.000,B 90.000,C 0.000} C_DIS
LIN {X -37.405,Y -28.575,Z -43.227,A -90.000,B 90.000,C 0.000} C_DIS
LIN {X -34.399,Y -28.575,Z -43.846,A -90.000,B 90.000,C 0.000} C_DIS
LIN {X -31.407,Y -28.575,Z -44.530,A -90.000,B 90.000,C 0.000} C_DIS
LIN {X -28.430,Y -28.575,Z -45.280,A -90.000,B 90.000,C 0.000} C_DIS
LIN {X -27.078,Y -28.575,Z -45.701,A -90.000,B 90.000,C 0.000} C_DIS
LIN {X -25.713,Y -28.575,Z -46.074,A -90.000,B 90.000,C 0.000} C_DIS
LIN {X -24.334,Y -28.575,Z -46.397,A -90.000,B 90.000,C 0.000} C_DIS
LIN {X -22.945,Y -28.575,Z -46.670,A -90.000,B 90.000,C 0.000} C_DIS
LIN {X -21.547,Y -28.575,Z -46.892,A -90.000,B 90.000,C 0.000} C_DIS
LIN {X -20.319,Y -28.575,Z -46.411,A -90.000,B 90.000,C 0.000} C_DIS
LIN {X -19.071,Y -28.575,Z -45.981,A -90.000,B 90.000,C 0.000} C_DIS
LIN {X -17.807,Y -28.575,Z -45.604,A -90.000,B 90.000,C 0.000} C_DIS
LIN {X -16.528,Y -28.575,Z -45.280,A -90.000,B 90.000,C 0.000} C_DIS
LIN {X -15.237,Y -28.575,Z -45.010,A -90.000,B 90.000,C 0.000} C_DIS
LIN {X -13.935,Y -28.575,Z -44.794,A -90.000,B 90.000,C 0.000} C_DIS
LIN {X -11.793,Y -28.575,Z -44.642,A -90.000,B 90.000,C 0.000} C_DIS
LIN {X -9.647,Y -28.575,Z -44.551,A -90.000,B 90.000,C 0.000} C_DIS
LIN {X -7.500,Y -28.575,Z -44.523,A -90.000,B 90.000,C 0.000} C_DIS
LIN {X -5.352,Y -28.575,Z -44.558,A -90.000,B 90.000,C 0.000} C_DIS
LIN {X -3.207,Y -28.575,Z -44.654,A -90.000,B 90.000,C 0.000} C_DIS
LIN {X -1.065,Y -28.575,Z -44.813,A -90.000,B 90.000,C 0.000} C_DIS
LIN {X 1.071,Y -28.575,Z -45.033,A -90.000,B 90.000,C 0.000} C_DIS
LIN {X 2.168,Y -28.575,Z -45.175,A -90.000,B 90.000,C 0.000} C_DIS
LIN {X 3.271,Y -28.575,Z -45.267,A -90.000,B 90.000,C 0.000} C_DIS
LIN {X 4.377,Y -28.575,Z -45.306,A -90.000,B 90.000,C 0.000} C_DIS
LIN {X 5.483,Y -28.575,Z -45.295,A -90.000,B 90.000,C 0.000} C_DIS
LIN {X 6.579,Y -28.575,Z -45.164,A -90.000,B 90.000,C 0.000} C_DIS
LIN {X 7.680,Y -28.575,Z -45.092,A -90.000,B 90.000,C 0.000} C_DIS
LIN {X 8.784,Y -28.575,Z -45.080,A -90.000,B 90.000,C 0.000} C_DIS
LIN {X 9.886,Y -28.575,Z -45.128,A -90.000,B 90.000,C 0.000} C_DIS
LIN {X 10.985,Y -28.575,Z -45.236,A -90.000,B 90.000,C 0.000} C_DIS
LIN {X 12.076,Y -28.575,Z -45.403,A -90.000,B 90.000,C 0.000} C_DIS
LIN {X 13.156,Y -28.575,Z -45.629,A -90.000,B 90.000,C 0.000} C_DIS
LIN {X 14.063,Y -28.575,Z -44.743,A -90.000,B 90.000,C 0.000} C_DIS
LIN {X 15.011,Y -28.575,Z -43.902,A -90.000,B 90.000,C 0.000} C_DIS
LIN {X 15.998,Y -28.575,Z -43.106,A -90.000,B 90.000,C 0.000} C_DIS
LIN {X 17.022,Y -28.575,Z -42.359,A -90.000,B 90.000,C 0.000} C_DIS
LIN {X 18.081,Y -28.575,Z -41.662,A -90.000,B 90.000,C 0.000} C_DIS
LIN {X 19.171,Y -28.575,Z -41.015,A -90.000,B 90.000,C 0.000} C_DIS
LIN {X 19.291,Y -28.575,Z -40.959,A -90.000,B 90.000,C 0.000} C_DIS
LIN {X 20.508,Y -28.575,Z -40.287,A -90.000,B 90.000,C 0.000} C_DIS
LIN {X 21.756,Y -28.575,Z -39.675,A -90.000,B 90.000,C 0.000} C_DIS
LIN {X 23.032,Y -28.575,Z -39.124,A -90.000,B 90.000,C 0.000} C_DIS
LIN {X 24.333,Y -28.575,Z -38.636,A -90.000,B 90.000,C 0.000} C_DIS
LIN {X 25.656,Y -28.575,Z -38.211,A -90.000,B 90.000,C 0.000} C_DIS
LIN {X 26.999,Y -28.575,Z -37.851,A -90.000,B 90.000,C 0.000} C_DIS
LIN {X 28.357,Y -28.575,Z -37.557,A -90.000,B 90.000,C 0.000} C_DIS
LIN {X 29.293,Y -28.575,Z -37.458,A -90.000,B 90.000,C 0.000} C_DIS
LIN {X 30.221,Y -28.575,Z -37.303,A -90.000,B 90.000,C 0.000} C_DIS
LIN {X 31.138,Y -28.575,Z -37.091,A -90.000,B 90.000,C 0.000} C_DIS
LIN {X 32.041,Y -28.575,Z -36.823,A -90.000,B 90.000,C 0.000} C_DIS
LIN {X 32.925,Y -28.575,Z -36.500,A -90.000,B 90.000,C 0.000} C_DIS
LIN {X 34.110,Y -28.575,Z -36.015,A -90.000,B 90.000,C 0.000} C_DIS
LIN {X 35.316,Y -28.575,Z -35.584,A -90.000,B 90.000,C 0.000} C_DIS
LIN {X 36.539,Y -28.575,Z -35.205,A -90.000,B 90.000,C 0.000} C_DIS
LIN {X 37.778,Y -28.575,Z -34.882,A -90.000,B 90.000,C 0.000} C_DIS
LIN {X 39.030,Y -28.575,Z -34.613,A -90.000,B 90.000,C 0.000} C_DIS
LIN {X 40.293,Y -28.575,Z -34.399,A -90.000,B 90.000,C 0.000} C_DIS
LIN {X 41.563,Y -28.575,Z -34.241,A -90.000,B 90.000,C 0.000} C_DIS
LIN {X 42.840,Y -28.575,Z -34.140,A -90.000,B 90.000,C 0.000} C_DIS
LIN {X 44.118,Y -28.575,Z -34.165,A -90.000,B 90.000,C 0.000} C_DIS
LIN {X 45.394,Y -28.575,Z -34.249,A -90.000,B 90.000,C 0.000} C_DIS
LIN {X 46.665,Y -28.575,Z -34.392,A -90.000,B 90.000,C 0.000} C_DIS
LIN {X 47.927,Y -28.575,Z -34.593,A -90.000,B 90.000,C 0.000} C_DIS
LIN {X 49.179,Y -28.575,Z -34.851,A -90.000,B 90.000,C 0.000} C_DIS
LIN {X 50.418,Y -28.575,Z -35.168,A -90.000,B 90.000,C 0.000} C_DIS
LIN {X 51.641,Y -28.575,Z -35.540,A -90.000,B 90.000,C 0.000} C_DIS
LIN {X 52.846,Y -28.575,Z -35.968,A -90.000,B 90.000,C 0.000} C_DIS
LIN {X 54.385,Y -28.575,Z -36.703,A -90.000,B 90.000,C 0.000} C_DIS
LIN {X 55.895,Y -28.575,Z -37.495,A -90.000,B 90.000,C 0.000} C_DIS
LIN {X 57.373,Y -28.575,Z -38.344,A -90.000,B 90.000,C 0.000} C_DIS
LIN {X 58.819,Y -28.575,Z -39.249,A -90.000,B 90.000,C 0.000} C_DIS
LIN {X 60.229,Y -28.575,Z -40.208,A -90.000,B 90.000,C 0.000} C_DIS
LIN {X 61.602,Y -28.575,Z -41.219,A -90.000,B 90.000,C 0.000} C_DIS
LIN {X 62.935,Y -28.575,Z -42.282,A -90.000,B 90.000,C 0.000} C_DIS
LIN {X 64.227,Y -28.575,Z -43.395,A -90.000,B 90.000,C 0.000} C_DIS
LIN {X 65.476,Y -28.575,Z -44.556,A -90.000,B 90.000,C 0.000} C_DIS
LIN {X 66.233,Y -28.575,Z -45.376,A -90.000,B 90.000,C 0.000} C_DIS
LIN {X 67.026,Y -28.575,Z -46.161,A -90.000,B 90.000,C 0.000} C_DIS
LIN {X 67.853,Y -28.575,Z -46.910,A -90.000,B 90.000,C 0.000} C_DIS
LIN {X 68.712,Y -28.575,Z -47.621,A -90.000,B 90.000,C 0.000} C_DIS
LIN {X 69.603,Y -28.575,Z -48.294,A -90.000,B 90.000,C 0.000} C_DIS
LIN {X 70.523,Y -28.575,Z -48.925,A -90.000,B 90.000,C 0.000} C_DIS
LIN {X 70.523,Y -41.075,Z -48.925,A -90.000,B 90.000,C 0.000} C_DIS
LIN {X 70.523,Y -53.575,Z -48.925,A -90.000,B 90.000,C 0.000} C_DIS
LIN {X 70.523,Y -54.260,Z -48.925,A -90.000,B 90.000,C 0.000} C_DIS
LIN {X -144.015,Y -54.260,Z -242.561,A -90.000,B 90.000,C 0.000} C_DIS
LIN {X -144.015,Y -46.431,Z -242.561,A -90.000,B 90.000,C 0.000} C_DIS
LIN {X -144.015,Y -33.931,Z -242.561,A -90.000,B 90.000,C 0.000} C_DIS
LIN {X -144.015,Y -21.431,Z -242.561,A -90.000,B 90.000,C 0.000} C_DIS
LIN {X -123.660,Y -21.431,Z -242.561,A -90.000,B 90.000,C 0.000} C_DIS
LIN {X -120.454,Y -21.431,Z -240.398,A -90.000,B 90.000,C 0.000} C_DIS
LIN {X -117.266,Y -21.431,Z -238.208,A -90.000,B 90.000,C 0.000} C_DIS
LIN {X -113.485,Y -21.431,Z -235.584,A -90.000,B 90.000,C 0.000} C_DIS
LIN {X -112.669,Y -21.431,Z -235.012,A -90.000,B 90.000,C 0.000} C_DIS
LIN {X -144.015,Y -21.431,Z -235.012,A -90.000,B 90.000,C 0.000} C_DIS
LIN {X -144.015,Y -21.431,Z -227.464,A -90.000,B 90.000,C 0.000} C_DIS
LIN {X -101.887,Y -21.431,Z -227.464,A -90.000,B 90.000,C 0.000} C_DIS
LIN {X -98.270,Y -21.431,Z -224.929,A -90.000,B 90.000,C 0.000} C_DIS
LIN {X -94.639,Y -21.431,Z -222.412,A -90.000,B 90.000,C 0.000} C_DIS
LIN {X -90.996,Y -21.431,Z -219.915,A -90.000,B 90.000,C 0.000} C_DIS
LIN {X -144.015,Y -21.431,Z -219.915,A -90.000,B 90.000,C 0.000} C_DIS
LIN {X -144.015,Y -21.431,Z -212.366,A -90.000,B 90.000,C 0.000} C_DIS
LIN {X -79.725,Y -21.431,Z -212.366,A -90.000,B 90.000,C 0.000} C_DIS
LIN {X -78.272,Y -21.431,Z -211.412,A -90.000,B 90.000,C 0.000} C_DIS
LIN {X -70.282,Y -21.431,Z -206.151,A -90.000,B 90.000,C 0.000} C_DIS
LIN {X -68.196,Y -21.431,Z -204.817,A -90.000,B 90.000,C 0.000} C_DIS
LIN {X -144.015,Y -21.431,Z -204.817,A -90.000,B 90.000,C 0.000} C_DIS
LIN {X -144.015,Y -21.431,Z -197.269,A -90.000,B 90.000,C 0.000} C_DIS
LIN {X -56.919,Y -21.431,Z -197.269,A -90.000,B 90.000,C 0.000} C_DIS
LIN {X -53.402,Y -21.431,Z -194.792,A -90.000,B 90.000,C 0.000} C_DIS
LIN {X -49.913,Y -21.431,Z -192.276,A -90.000,B 90.000,C 0.000} C_DIS
LIN {X -46.453,Y -21.431,Z -189.720,A -90.000,B 90.000,C 0.000} C_DIS
LIN {X -144.015,Y -21.431,Z -189.720,A -90.000,B 90.000,C 0.000} C_DIS
LIN {X -144.015,Y -21.431,Z -182.171,A -90.000,B 90.000,C 0.000} C_DIS
LIN {X -36.688,Y -21.431,Z -182.171,A -90.000,B 90.000,C 0.000} C_DIS
LIN {X -36.091,Y -21.431,Z -181.692,A -90.000,B 90.000,C 0.000} C_DIS
LIN {X -34.649,Y -21.431,Z -180.605,A -90.000,B 90.000,C 0.000} C_DIS
LIN {X -33.237,Y -21.431,Z -179.480,A -90.000,B 90.000,C 0.000} C_DIS
LIN {X -31.854,Y -21.431,Z -178.318,A -90.000,B 90.000,C 0.000} C_DIS
LIN {X -30.502,Y -21.431,Z -177.121,A -90.000,B 90.000,C 0.000} C_DIS
LIN {X -29.182,Y -21.431,Z -175.889,A -90.000,B 90.000,C 0.000} C_DIS
LIN {X -27.895,Y -21.431,Z -174.622,A -90.000,B 90.000,C 0.000} C_DIS
LIN {X -144.015,Y -21.431,Z -174.622,A -90.000,B 90.000,C 0.000} C_DIS
LIN {X -144.015,Y -21.431,Z -167.073,A -90.000,B 90.000,C 0.000} C_DIS
LIN {X -21.483,Y -21.431,Z -167.073,A -90.000,B 90.000,C 0.000} C_DIS
LIN {X -20.818,Y -21.431,Z -165.982,A -90.000,B 90.000,C 0.000} C_DIS
LIN {X -20.201,Y -21.431,Z -164.864,A -90.000,B 90.000,C 0.000} C_DIS
LIN {X -19.631,Y -21.431,Z -163.721,A -90.000,B 90.000,C 0.000} C_DIS
LIN {X -19.813,Y -21.431,Z -163.514,A -90.000,B 90.000,C 0.000} C_DIS
LIN {X -19.887,Y -21.431,Z -163.416,A -90.000,B 90.000,C 0.000} C_DIS
LIN {X -20.611,Y -21.431,Z -162.661,A -90.000,B 90.000,C 0.000} C_DIS
LIN {X -21.363,Y -21.431,Z -161.935,A -90.000,B 90.000,C 0.000} C_DIS
LIN {X -22.694,Y -21.431,Z -160.733,A -90.000,B 90.000,C 0.000} C_DIS
LIN {X -24.019,Y -21.431,Z -159.525,A -90.000,B 90.000,C 0.000} C_DIS
LIN {X -144.015,Y -21.431,Z -159.525,A -90.000,B 90.000,C 0.000} C_DIS
LIN {X -144.015,Y -21.431,Z -151.976,A -90.000,B 90.000,C 0.000} C_DIS
LIN {X -32.062,Y -21.431,Z -151.976,A -90.000,B 90.000,C 0.000} C_DIS
LIN {X -33.208,Y -21.431,Z -150.793,A -90.000,B 90.000,C 0.000} C_DIS
LIN {X -34.322,Y -21.431,Z -149.578,A -90.000,B 90.000,C 0.000} C_DIS
LIN {X -35.401,Y -21.431,Z -148.333,A -90.000,B 90.000,C 0.000} C_DIS
LIN {X -36.445,Y -21.431,Z -147.059,A -90.000,B 90.000,C 0.000} C_DIS
LIN {X -37.454,Y -21.431,Z -145.757,A -90.000,B 90.000,C 0.000} C_DIS
LIN {X -38.427,Y -21.431,Z -144.427,A -90.000,B 90.000,C 0.000} C_DIS
LIN {X -144.015,Y -21.431,Z -144.427,A -90.000,B 90.000,C 0.000} C_DIS
LIN {X -144.015,Y -21.431,Z -136.878,A -90.000,B 90.000,C 0.000} C_DIS
LIN {X -42.841,Y -21.431,Z -136.878,A -90.000,B 90.000,C 0.000} C_DIS
LIN {X -43.764,Y -21.431,Z -135.024,A -90.000,B 90.000,C 0.000} C_DIS
LIN {X -44.639,Y -21.431,Z -133.147,A -90.000,B 90.000,C 0.000} C_DIS
LIN {X -45.466,Y -21.431,Z -131.248,A -90.000,B 90.000,C 0.000} C_DIS
LIN {X -46.244,Y -21.431,Z -129.329,A -90.000,B 90.000,C 0.000} C_DIS
LIN {X -144.015,Y -21.431,Z -129.329,A -90.000,B 90.000,C 0.000} C_DIS
LIN {X -144.015,Y -21.431,Z -121.781,A -90.000,B 90.000,C 0.000} C_DIS
LIN {X -50.508,Y -21.431,Z -121.781,A -90.000,B 90.000,C 0.000} C_DIS
LIN {X -52.549,Y -21.431,Z -119.290,A -90.000,B 90.000,C 0.000} C_DIS
LIN {X -54.558,Y -21.431,Z -116.773,A -90.000,B 90.000,C 0.000} C_DIS
LIN {X -56.537,Y -21.431,Z -114.232,A -90.000,B 90.000,C 0.000} C_DIS
LIN {X -144.015,Y -21.431,Z -114.232,A -90.000,B 90.000,C 0.000} C_DIS
LIN {X -144.015,Y -21.431,Z -106.683,A -90.000,B 90.000,C 0.000} C_DIS
LIN {X -62.127,Y -21.431,Z -106.683,A -90.000,B 90.000,C 0.000} C_DIS
LIN {X -63.648,Y -21.431,Z -104.572,A -90.000,B 90.000,C 0.000} C_DIS
LIN {X -65.192,Y -21.431,Z -102.477,A -90.000,B 90.000,C 0.000} C_DIS
LIN {X -66.010,Y -21.431,Z -101.349,A -90.000,B 90.000,C 0.000} C_DIS
LIN {X -66.847,Y -21.431,Z -100.235,A -90.000,B 90.000,C 0.000} C_DIS
LIN {X -67.701,Y -21.431,Z -99.134,A -90.000,B 90.000,C 0.000} C_DIS
LIN {X -144.015,Y -21.431,Z -99.134,A -90.000,B 90.000,C 0.000} C_DIS
LIN {X -144.015,Y -21.431,Z -91.586,A -90.000,B 90.000,C 0.000} C_DIS
LIN {X -74.431,Y -21.431,Z -91.586,A -90.000,B 90.000,C 0.000} C_DIS
LIN {X -75.781,Y -21.431,Z -90.272,A -90.000,B 90.000,C 0.000} C_DIS
LIN {X -77.159,Y -21.431,Z -88.988,A -90.000,B 90.000,C 0.000} C_DIS
LIN {X -77.660,Y -21.431,Z -88.474,A -90.000,B 90.000,C 0.000} C_DIS
LIN {X -78.205,Y -21.431,Z -88.006,A -90.000,B 90.000,C 0.000} C_DIS
LIN {X -78.789,Y -21.431,Z -87.589,A -90.000,B 90.000,C 0.000} C_DIS
LIN {X -79.408,Y -21.431,Z -87.226,A -90.000,B 90.000,C 0.000} C_DIS
LIN {X -80.057,Y -21.431,Z -86.919,A -90.000,B 90.000,C 0.000} C_DIS
LIN {X -81.393,Y -21.431,Z -86.450,A -90.000,B 90.000,C 0.000} C_DIS
LIN {X -82.709,Y -21.431,Z -85.926,A -90.000,B 90.000,C 0.000} C_DIS
LIN {X -84.002,Y -21.431,Z -85.349,A -90.000,B 90.000,C 0.000} C_DIS
LIN {X -85.270,Y -21.431,Z -84.719,A -90.000,B 90.000,C 0.000} C_DIS
LIN {X -86.511,Y -21.431,Z -84.037,A -90.000,B 90.000,C 0.000} C_DIS
LIN {X -144.015,Y -21.431,Z -84.037,A -90.000,B 90.000,C 0.000} C_DIS
LIN {X -144.015,Y -21.431,Z -76.488,A -90.000,B 90.000,C 0.000} C_DIS
LIN {X -96.953,Y -21.431,Z -76.488,A -90.000,B 90.000,C 0.000} C_DIS
LIN {X -98.495,Y -21.431,Z -75.540,A -90.000,B 90.000,C 0.000} C_DIS
LIN {X -100.008,Y -21.431,Z -74.547,A -90.000,B 90.000,C 0.000} C_DIS
LIN {X -101.491,Y -21.431,Z -73.510,A -90.000,B 90.000,C 0.000} C_DIS
LIN {X -102.944,Y -21.431,Z -72.429,A -90.000,B 90.000,C 0.000} C_DIS
LIN {X -104.364,Y -21.431,Z -71.307,A -90.000,B 90.000,C 0.000} C_DIS
LIN {X -105.750,Y -21.431,Z -70.143,A -90.000,B 90.000,C 0.000} C_DIS
LIN {X -107.101,Y -21.431,Z -68.939,A -90.000,B 90.000,C 0.000} C_DIS
LIN {X -144.015,Y -21.431,Z -68.939,A -90.000,B 90.000,C 0.000} C_DIS
LIN {X -144.015,Y -21.431,Z -61.390,A -90.000,B 90.000,C 0.000} C_DIS
LIN {X -114.090,Y -21.431,Z -61.390,A -90.000,B 90.000,C 0.000} C_DIS
LIN {X -114.704,Y -21.431,Z -60.488,A -90.000,B 90.000,C 0.000} C_DIS
LIN {X -115.262,Y -21.431,Z -59.551,A -90.000,B 90.000,C 0.000} C_DIS
LIN {X -115.762,Y -21.431,Z -58.582,A -90.000,B 90.000,C 0.000} C_DIS
LIN {X -116.203,Y -21.431,Z -57.585,A -90.000,B 90.000,C 0.000} C_DIS
LIN {X -116.583,Y -21.431,Z -56.562,A -90.000,B 90.000,C 0.000} C_DIS
LIN {X -116.900,Y -21.431,Z -55.519,A -90.000,B 90.000,C 0.000} C_DIS
LIN {X -117.084,Y -21.431,Z -54.967,A -90.000,B 90.000,C 0.000} C_DIS
LIN {X -117.243,Y -21.431,Z -54.408,A -90.000,B 90.000,C 0.000} C_DIS
LIN {X -117.379,Y -21.431,Z -53.842,A -90.000,B 90.000,C 0.000} C_DIS
LIN {X -144.015,Y -21.431,Z -53.842,A -90.000,B 90.000,C 0.000} C_DIS
LIN {X -144.015,Y -21.431,Z -46.293,A -90.000,B 90.000,C 0.000} C_DIS
LIN {X -118.053,Y -21.431,Z -46.293,A -90.000,B 90.000,C 0.000} C_DIS
LIN {X -118.290,Y -21.431,Z -45.268,A -90.000,B 90.000,C 0.000} C_DIS
LIN {X -118.463,Y -21.431,Z -44.231,A -90.000,B 90.000,C 0.000} C_DIS
LIN {X -118.571,Y -21.431,Z -43.184,A -90.000,B 90.000,C 0.000} C_DIS
LIN {X -118.612,Y -21.431,Z -42.133,A -90.000,B 90.000,C 0.000} C_DIS
LIN {X -118.588,Y -21.431,Z -41.082,A -90.000,B 90.000,C 0.000} C_DIS
LIN {X -118.497,Y -21.431,Z -40.034,A -90.000,B 90.000,C 0.000} C_DIS
LIN {X -118.470,Y -21.431,Z -39.854,A -90.000,B 90.000,C 0.000} C_DIS
LIN {X -118.380,Y -21.431,Z -39.297,A -90.000,B 90.000,C 0.000} C_DIS
LIN {X -118.269,Y -21.431,Z -38.744,A -90.000,B 90.000,C 0.000} C_DIS
LIN {X -144.015,Y -21.431,Z -38.744,A -90.000,B 90.000,C 0.000} C_DIS
LIN {X -144.015,Y -21.431,Z -31.195,A -90.000,B 90.000,C 0.000} C_DIS
LIN {X -113.849,Y -21.431,Z -31.195,A -90.000,B 90.000,C 0.000} C_DIS
LIN {X -112.962,Y -21.431,Z -30.468,A -90.000,B 90.000,C 0.000} C_DIS
LIN {X -112.853,Y -21.431,Z -30.393,A -90.000,B 90.000,C 0.000} C_DIS
LIN {X -112.377,Y -21.431,Z -30.059,A -90.000,B 90.000,C 0.000} C_DIS
LIN {X -111.881,Y -21.431,Z -29.755,A -90.000,B 90.000,C 0.000} C_DIS
LIN {X -111.368,Y -21.431,Z -29.482,A -90.000,B 90.000,C 0.000} C_DIS
LIN {X -110.840,Y -21.431,Z -29.239,A -90.000,B 90.000,C 0.000} C_DIS
LIN {X -109.927,Y -21.431,Z -28.433,A -90.000,B 90.000,C 0.000} C_DIS
LIN {X -108.977,Y -21.431,Z -27.671,A -90.000,B 90.000,C 0.000} C_DIS
LIN {X -107.993,Y -21.431,Z -26.953,A -90.000,B 90.000,C 0.000} C_DIS
LIN {X -106.977,Y -21.431,Z -26.282,A -90.000,B 90.000,C 0.000} C_DIS
LIN {X -105.931,Y -21.431,Z -25.658,A -90.000,B 90.000,C 0.000} C_DIS
LIN {X -105.556,Y -21.431,Z -24.965,A -90.000,B 90.000,C 0.000} C_DIS
LIN {X -105.145,Y -21.431,Z -24.294,A -90.000,B 90.000,C 0.000} C_DIS
LIN {X -104.697,Y -21.431,Z -23.646,A -90.000,B 90.000,C 0.000} C_DIS
LIN {X -144.015,Y -21.431,Z -23.646,A -90.000,B 90.000,C 0.000} C_DIS
LIN {X -144.015,Y -21.431,Z -16.098,A -90.000,B 90.000,C 0.000} C_DIS
LIN {X -91.772,Y -21.431,Z -16.098,A -90.000,B 90.000,C 0.000} C_DIS
LIN {X -91.394,Y -21.431,Z -15.403,A -90.000,B 90.000,C 0.000} C_DIS
LIN {X -90.976,Y -21.431,Z -14.730,A -90.000,B 90.000,C 0.000} C_DIS
LIN {X -90.522,Y -21.431,Z -14.083,A -90.000,B 90.000,C 0.000} C_DIS
LIN {X -90.032,Y -21.431,Z -13.462,A -90.000,B 90.000,C 0.000} C_DIS
LIN {X -89.507,Y -21.431,Z -12.869,A -90.000,B 90.000,C 0.000} C_DIS
LIN {X -88.743,Y -21.431,Z -12.165,A -90.000,B 90.000,C 0.000} C_DIS
LIN {X -87.936,Y -21.431,Z -11.512,A -90.000,B 90.000,C 0.000} C_DIS
LIN {X -87.088,Y -21.431,Z -10.912,A -90.000,B 90.000,C 0.000} C_DIS
LIN {X -86.204,Y -21.431,Z -10.367,A -90.000,B 90.000,C 0.000} C_DIS
LIN {X -85.287,Y -21.431,Z -9.880,A -90.000,B 90.000,C 0.000} C_DIS
LIN {X -84.340,Y -21.431,Z -9.454,A -90.000,B 90.000,C 0.000} C_DIS
LIN {X -83.368,Y -21.431,Z -9.088,A -90.000,B 90.000,C 0.000} C_DIS
LIN {X -82.374,Y -21.431,Z -8.786,A -90.000,B 90.000,C 0.000} C_DIS
LIN {X -81.363,Y -21.431,Z -8.549,A -90.000,B 90.000,C 0.000} C_DIS
LIN {X -144.015,Y -21.431,Z -8.549,A -90.000,B 90.000,C 0.000} C_DIS
LIN {X -144.015,Y -21.431,Z -1.000,A -90.000,B 90.000,C 0.000} C_DIS
LIN {X 144.015,Y -21.431,Z -1.000,A -90.000,B 90.000,C 0.000} C_DIS
LIN {X 144.015,Y -21.431,Z -8.549,A -90.000,B 90.000,C 0.000} C_DIS
LIN {X -75.451,Y -21.431,Z -8.549,A -90.000,B 90.000,C 0.000} C_DIS
LIN {X -74.264,Y -21.431,Z -8.777,A -90.000,B 90.000,C 0.000} C_DIS
LIN {X -73.091,Y -21.431,Z -9.064,A -90.000,B 90.000,C 0.000} C_DIS
LIN {X -71.933,Y -21.431,Z -9.410,A -90.000,B 90.000,C 0.000} C_DIS
LIN {X -70.794,Y -21.431,Z -9.814,A -90.000,B 90.000,C 0.000} C_DIS
LIN {X -69.677,Y -21.431,Z -10.275,A -90.000,B 90.000,C 0.000} C_DIS
LIN {X -68.585,Y -21.431,Z -10.791,A -90.000,B 90.000,C 0.000} C_DIS
LIN {X -67.442,Y -21.431,Z -11.388,A -90.000,B 90.000,C 0.000} C_DIS
LIN {X -66.330,Y -21.431,Z -12.042,A -90.000,B 90.000,C 0.000} C_DIS
LIN {X -65.252,Y -21.431,Z -12.751,A -90.000,B 90.000,C 0.000} C_DIS
LIN {X -64.211,Y -21.431,Z -13.513,A -90.000,B 90.000,C 0.000} C_DIS
LIN {X -63.210,Y -21.431,Z -14.326,A -90.000,B 90.000,C 0.000} C_DIS
LIN {X -62.251,Y -21.431,Z -15.188,A -90.000,B 90.000,C 0.000} C_DIS
LIN {X -61.336,Y -21.431,Z -16.098,A -90.000,B 90.000,C 0.000} C_DIS
LIN {X 144.015,Y -21.431,Z -16.098,A -90.000,B 90.000,C 0.000} C_DIS
LIN {X 144.015,Y -21.431,Z -23.646,A -90.000,B 90.000,C 0.000} C_DIS
LIN {X -50.835,Y -21.431,Z -23.646,A -90.000,B 90.000,C 0.000} C_DIS
LIN {X -50.288,Y -21.431,Z -23.692,A -90.000,B 90.000,C 0.000} C_DIS
LIN {X -49.740,Y -21.431,Z -23.730,A -90.000,B 90.000,C 0.000} C_DIS
LIN {X -49.625,Y -21.431,Z -23.735,A -90.000,B 90.000,C 0.000} C_DIS
LIN {X -48.795,Y -21.431,Z -23.706,A -90.000,B 90.000,C 0.000} C_DIS
LIN {X -47.965,Y -21.431,Z -23.721,A -90.000,B 90.000,C 0.000} C_DIS
LIN {X -47.136,Y -21.431,Z -23.780,A -90.000,B 90.000,C 0.000} C_DIS
LIN {X -46.312,Y -21.431,Z -23.884,A -90.000,B 90.000,C 0.000} C_DIS
LIN {X -43.239,Y -21.431,Z -23.942,A -90.000,B 90.000,C 0.000} C_DIS
LIN {X -40.169,Y -21.431,Z -24.066,A -90.000,B 90.000,C 0.000} C_DIS
LIN {X -37.101,Y -21.431,Z -24.257,A -90.000,B 90.000,C 0.000} C_DIS
LIN {X -34.039,Y -21.431,Z -24.514,A -90.000,B 90.000,C 0.000} C_DIS
LIN {X -30.983,Y -21.431,Z -24.837,A -90.000,B 90.000,C 0.000} C_DIS
LIN {X -27.934,Y -21.431,Z -25.226,A -90.000,B 90.000,C 0.000} C_DIS
LIN {X -24.895,Y -21.431,Z -25.681,A -90.000,B 90.000,C 0.000} C_DIS
LIN {X -21.866,Y -21.431,Z -26.202,A -90.000,B 90.000,C 0.000} C_DIS
LIN {X -18.849,Y -21.431,Z -26.787,A -90.000,B 90.000,C 0.000} C_DIS
LIN {X -15.845,Y -21.431,Z -27.438,A -90.000,B 90.000,C 0.000} C_DIS
LIN {X -12.857,Y -21.431,Z -28.154,A -90.000,B 90.000,C 0.000} C_DIS
LIN {X -9.884,Y -21.431,Z -28.934,A -90.000,B 90.000,C 0.000} C_DIS
LIN {X -6.929,Y -21.431,Z -29.778,A -90.000,B 90.000,C 0.000} C_DIS
LIN {X -6.050,Y -21.431,Z -30.083,A -90.000,B 90.000,C 0.000} C_DIS
LIN {X -5.161,Y -21.431,Z -30.356,A -90.000,B 90.000,C 0.000} C_DIS
LIN {X -4.261,Y -21.431,Z -30.594,A -90.000,B 90.000,C 0.000} C_DIS
LIN {X -3.354,Y -21.431,Z -30.799,A -90.000,B 90.000,C 0.000} C_DIS
LIN {X -0.725,Y -21.431,Z -31.195,A -90.000,B 90.000,C 0.000} C_DIS
LIN {X 28.405,Y -21.431,Z -31.195,A -90.000,B 90.000,C 0.000} C_DIS
LIN {X 30.879,Y -21.431,Z -30.837,A -90.000,B 90.000,C 0.000} C_DIS
LIN {X 33.358,Y -21.431,Z -30.519,A -90.000,B 90.000,C 0.000} C_DIS
LIN {X 34.958,Y -21.431,Z -30.434,A -90.000,B 90.000,C 0.000} C_DIS
LIN {X 36.560,Y -21.431,Z -30.410,A -90.000,B 90.000,C 0.000} C_DIS
LIN {X 38.161,Y -21.431,Z -30.447,A -90.000,B 90.000,C 0.000} C_DIS
LIN {X 39.760,Y -21.431,Z -30.544,A -90.000,B 90.000,C 0.000} C_DIS
LIN {X 41.355,Y -21.431,Z -30.701,A -90.000,B 90.000,C 0.000} C_DIS
LIN {X 42.942,Y -21.431,Z -30.918,A -90.000,B 90.000,C 0.000} C_DIS
LIN {X 44.520,Y -21.431,Z -31.195,A -90.000,B 90.000,C 0.000} C_DIS
LIN {X 98.289,Y -21.431,Z -31.195,A -90.000,B 90.000,C 0.000} C_DIS
LIN {X 96.315,Y -21.431,Z -32.157,A -90.000,B 90.000,C 0.000} C_DIS
LIN {X 94.368,Y -21.431,Z -33.171,A -90.000,B 90.000,C 0.000} C_DIS
LIN {X 92.448,Y -21.431,Z -34.238,A -90.000,B 90.000,C 0.000} C_DIS
LIN {X 90.558,Y -21.431,Z -35.355,A -90.000,B 90.000,C 0.000} C_DIS
LIN {X 88.699,Y -21.431,Z -36.523,A -90.000,B 90.000,C 0.000} C_DIS
LIN {X 87.662,Y -21.431,Z -37.232,A -90.000,B 90.000,C 0.000} C_DIS
LIN {X 86.648,Y -21.431,Z -37.973,A -90.000,B 90.000,C 0.000} C_DIS
LIN {X 85.657,Y -21.431,Z -38.744,A -90.000,B 90.000,C 0.000} C_DIS
LIN {X 60.643,Y -21.431,Z -38.744,A -90.000,B 90.000,C 0.000} C_DIS
LIN {X 61.560,Y -21.431,Z -39.417,A -90.000,B 90.000,C 0.000} C_DIS
LIN {X 62.462,Y -21.431,Z -40.111,A -90.000,B 90.000,C 0.000} C_DIS
LIN {X 63.474,Y -21.431,Z -41.051,A -90.000,B 90.000,C 0.000} C_DIS
LIN {X 64.517,Y -21.431,Z -41.957,A -90.000,B 90.000,C 0.000} C_DIS
LIN {X 65.590,Y -21.431,Z -42.826,A -90.000,B 90.000,C 0.000} C_DIS
LIN {X 66.692,Y -21.431,Z -43.658,A -90.000,B 90.000,C 0.000} C_DIS
LIN {X 67.821,Y -21.431,Z -44.453,A -90.000,B 90.000,C 0.000} C_DIS
LIN {X 68.977,Y -21.431,Z -45.209,A -90.000,B 90.000,C 0.000} C_DIS
LIN {X 70.001,Y -21.431,Z -45.744,A -90.000,B 90.000,C 0.000} C_DIS
LIN {X 71.017,Y -21.431,Z -46.293,A -90.000,B 90.000,C 0.000} C_DIS
LIN {X 78.400,Y -21.431,Z -46.293,A -90.000,B 90.000,C 0.000} C_DIS
LIN {X 79.368,Y -21.431,Z -45.037,A -90.000,B 90.000,C 0.000} C_DIS
LIN {X 80.384,Y -21.431,Z -43.820,A -90.000,B 90.000,C 0.000} C_DIS
LIN {X 81.446,Y -21.431,Z -42.644,A -90.000,B 90.000,C 0.000} C_DIS
LIN {X 82.553,Y -21.431,Z -41.509,A -90.000,B 90.000,C 0.000} C_DIS
LIN {X 83.703,Y -21.431,Z -40.418,A -90.000,B 90.000,C 0.000} C_DIS
LIN {X 84.894,Y -21.431,Z -39.372,A -90.000,B 90.000,C 0.000} C_DIS
LIN {X 86.125,Y -21.431,Z -38.373,A -90.000,B 90.000,C 0.000} C_DIS
LIN {X 87.394,Y -21.431,Z -37.423,A -90.000,B 90.000,C 0.000} C_DIS
LIN {X 88.699,Y -21.431,Z -36.523,A -90.000,B 90.000,C 0.000} C_DIS
LIN {X 90.540,Y -21.431,Z -35.367,A -90.000,B 90.000,C 0.000} C_DIS
LIN {X 92.411,Y -21.431,Z -34.260,A -90.000,B 90.000,C 0.000} C_DIS
LIN {X 94.310,Y -21.431,Z -33.203,A -90.000,B 90.000,C 0.000} C_DIS
LIN {X 96.237,Y -21.431,Z -32.197,A -90.000,B 90.000,C 0.000} C_DIS
LIN {X 98.190,Y -21.431,Z -31.242,A -90.000,B 90.000,C 0.000} C_DIS
LIN {X 100.168,Y -21.431,Z -30.339,A -90.000,B 90.000,C 0.000} C_DIS
LIN {X 102.168,Y -21.431,Z -29.490,A -90.000,B 90.000,C 0.000} C_DIS
LIN {X 104.191,Y -21.431,Z -28.693,A -90.000,B 90.000,C 0.000} C_DIS
LIN {X 105.133,Y -21.431,Z -28.307,A -90.000,B 90.000,C 0.000} C_DIS
LIN {X 106.098,Y -21.431,Z -27.984,A -90.000,B 90.000,C 0.000} C_DIS
LIN {X 107.083,Y -21.431,Z -27.726,A -90.000,B 90.000,C 0.000} C_DIS
LIN {X 108.083,Y -21.431,Z -27.534,A -90.000,B 90.000,C 0.000} C_DIS
LIN {X 109.093,Y -21.431,Z -27.409,A -90.000,B 90.000,C 0.000} C_DIS
LIN {X 110.109,Y -21.431,Z -27.351,A -90.000,B 90.000,C 0.000} C_DIS
LIN {X 111.127,Y -21.431,Z -27.360,A -90.000,B 90.000,C 0.000} C_DIS
LIN {X 112.142,Y -21.431,Z -27.436,A -90.000,B 90.000,C 0.000} C_DIS
LIN {X 113.150,Y -21.431,Z -27.580,A -90.000,B 90.000,C 0.000} C_DIS
LIN {X 114.146,Y -21.431,Z -27.790,A -90.000,B 90.000,C 0.000} C_DIS
LIN {X 115.126,Y -21.431,Z -28.066,A -90.000,B 90.000,C 0.000} C_DIS
LIN {X 116.085,Y -21.431,Z -28.406,A -90.000,B 90.000,C 0.000} C_DIS
LIN {X 117.020,Y -21.431,Z -28.809,A -90.000,B 90.000,C 0.000} C_DIS
LIN {X 117.926,Y -21.431,Z -29.273,A -90.000,B 90.000,C 0.000} C_DIS
LIN {X 118.799,Y -21.431,Z -29.796,A -90.000,B 90.000,C 0.000} C_DIS
LIN {X 119.636,Y -21.431,Z -30.376,A -90.000,B 90.000,C 0.000} C_DIS
LIN {X 119.758,Y -21.431,Z -30.472,A -90.000,B 90.000,C 0.000} C_DIS
LIN {X 120.185,Y -21.431,Z -30.827,A -90.000,B 90.000,C 0.000} C_DIS
LIN {X 120.600,Y -21.431,Z -31.195,A -90.000,B 90.000,C 0.000} C_DIS
LIN {X 144.015,Y -21.431,Z -31.195,A -90.000,B 90.000,C 0.000} C_DIS
LIN {X 144.015,Y -21.431,Z -38.744,A -90.000,B 90.000,C 0.000} C_DIS
LIN {X 124.956,Y -21.431,Z -38.744,A -90.000,B 90.000,C 0.000} C_DIS
LIN {X 125.148,Y -21.431,Z -39.640,A -90.000,B 90.000,C 0.000} C_DIS
LIN {X 125.291,Y -21.431,Z -40.545,A -90.000,B 90.000,C 0.000} C_DIS
LIN {X 125.384,Y -21.431,Z -41.456,A -90.000,B 90.000,C 0.000} C_DIS
LIN {X 125.427,Y -21.431,Z -42.371,A -90.000,B 90.000,C 0.000} C_DIS
LIN {X 125.420,Y -21.431,Z -43.288,A -90.000,B 90.000,C 0.000} C_DIS
LIN {X 125.363,Y -21.431,Z -44.202,A -90.000,B 90.000,C 0.000} C_DIS
LIN {X 125.205,Y -21.431,Z -45.251,A -90.000,B 90.000,C 0.000} C_DIS
LIN {X 125.008,Y -21.431,Z -46.293,A -90.000,B 90.000,C 0.000} C_DIS
LIN {X 144.015,Y -21.431,Z -46.293,A -90.000,B 90.000,C 0.000} C_DIS
LIN {X 144.015,Y -21.431,Z -53.842,A -90.000,B 90.000,C 0.000} C_DIS
LIN {X 122.255,Y -21.431,Z -53.842,A -90.000,B 90.000,C 0.000} C_DIS
LIN {X 121.608,Y -21.431,Z -55.049,A -90.000,B 90.000,C 0.000} C_DIS
LIN {X 121.005,Y -21.431,Z -56.278,A -90.000,B 90.000,C 0.000} C_DIS
LIN {X 120.448,Y -21.431,Z -57.529,A -90.000,B 90.000,C 0.000} C_DIS
LIN {X 119.936,Y -21.431,Z -58.799,A -90.000,B 90.000,C 0.000} C_DIS
LIN {X 119.470,Y -21.431,Z -60.086,A -90.000,B 90.000,C 0.000} C_DIS
LIN {X 119.052,Y -21.431,Z -61.390,A -90.000,B 90.000,C 0.000} C_DIS
LIN {X 144.015,Y -21.431,Z -61.390,A -90.000,B 90.000,C 0.000} C_DIS
LIN {X 144.015,Y -21.431,Z -68.939,A -90.000,B 90.000,C 0.000} C_DIS
LIN {X 116.946,Y -21.431,Z -68.939,A -90.000,B 90.000,C 0.000} C_DIS
LIN {X 116.289,Y -21.431,Z -70.855,A -90.000,B 90.000,C 0.000} C_DIS
LIN {X 115.581,Y -21.431,Z -72.752,A -90.000,B 90.000,C 0.000} C_DIS
LIN {X 114.823,Y -21.431,Z -74.631,A -90.000,B 90.000,C 0.000} C_DIS
LIN {X 114.015,Y -21.431,Z -76.488,A -90.000,B 90.000,C 0.000} C_DIS
LIN {X 144.015,Y -21.431,Z -76.488,A -90.000,B 90.000,C 0.000} C_DIS
LIN {X 144.015,Y -21.431,Z -84.037,A -90.000,B 90.000,C 0.000} C_DIS
LIN {X 110.095,Y -21.431,Z -84.037,A -90.000,B 90.000,C 0.000} C_DIS
LIN {X 109.309,Y -21.431,Z -85.334,A -90.000,B 90.000,C 0.000} C_DIS
LIN {X 108.498,Y -21.431,Z -86.615,A -90.000,B 90.000,C 0.000} C_DIS
LIN {X 107.661,Y -21.431,Z -87.880,A -90.000,B 90.000,C 0.000} C_DIS
LIN {X 107.686,Y -21.431,Z -88.238,A -90.000,B 90.000,C 0.000} C_DIS
LIN {X 107.984,Y -21.431,Z -89.060,A -90.000,B 90.000,C 0.000} C_DIS
LIN {X 108.250,Y -21.431,Z -89.893,A -90.000,B 90.000,C 0.000} C_DIS
LIN {X 108.484,Y -21.431,Z -90.735,A -90.000,B 90.000,C 0.000} C_DIS
LIN {X 108.686,Y -21.431,Z -91.586,A -90.000,B 90.000,C 0.000} C_DIS
LIN {X 144.015,Y -21.431,Z -91.586,A -90.000,B 90.000,C 0.000} C_DIS
LIN {X 144.015,Y -21.431,Z -99.134,A -90.000,B 90.000,C 0.000} C_DIS
LIN {X 109.863,Y -21.431,Z -99.134,A -90.000,B 90.000,C 0.000} C_DIS
LIN {X 110.073,Y -21.431,Z -100.576,A -90.000,B 90.000,C 0.000} C_DIS
LIN {X 110.299,Y -21.431,Z -102.016,A -90.000,B 90.000,C 0.000} C_DIS
LIN {X 110.695,Y -21.431,Z -104.347,A -90.000,B 90.000,C 0.000} C_DIS
LIN {X 111.064,Y -21.431,Z -106.683,A -90.000,B 90.000,C 0.000} C_DIS
LIN {X 144.015,Y -21.431,Z -106.683,A -90.000,B 90.000,C 0.000} C_DIS
LIN {X 144.015,Y -21.431,Z -114.232,A -90.000,B 90.000,C 0.000} C_DIS
LIN {X 112.069,Y -21.431,Z -114.232,A -90.000,B 90.000,C 0.000} C_DIS
LIN {X 112.340,Y -21.431,Z -116.745,A -90.000,B 90.000,C 0.000} C_DIS
LIN {X 112.580,Y -21.431,Z -119.262,A -90.000,B 90.000,C 0.000} C_DIS
LIN {X 112.789,Y -21.431,Z -121.781,A -90.000,B 90.000,C 0.000} C_DIS
LIN {X 144.015,Y -21.431,Z -121.781,A -90.000,B 90.000,C 0.000} C_DIS
LIN {X 144.015,Y -21.431,Z -129.329,A -90.000,B 90.000,C 0.000} C_DIS
LIN {X 113.227,Y -21.431,Z -129.329,A -90.000,B 90.000,C 0.000} C_DIS
LIN {X 113.232,Y -21.431,Z -129.470,A -90.000,B 90.000,C 0.000} C_DIS
LIN {X 113.220,Y -21.431,Z -133.174,A -90.000,B 90.000,C 0.000} C_DIS
LIN {X 113.162,Y -21.431,Z -136.878,A -90.000,B 90.000,C 0.000} C_DIS
LIN {X 144.015,Y -21.431,Z -136.878,A -90.000,B 90.000,C 0.000} C_DIS
LIN {X 144.015,Y -21.431,Z -144.427,A -90.000,B 90.000,C 0.000} C_DIS
LIN {X 112.905,Y -21.431,Z -144.427,A -90.000,B 90.000,C 0.000} C_DIS
LIN {X 112.778,Y -21.431,Z -146.945,A -90.000,B 90.000,C 0.000} C_DIS
LIN {X 112.629,Y -21.431,Z -149.461,A -90.000,B 90.000,C 0.000} C_DIS
LIN {X 112.461,Y -21.431,Z -151.976,A -90.000,B 90.000,C 0.000} C_DIS
LIN {X 144.015,Y -21.431,Z -151.976,A -90.000,B 90.000,C 0.000} C_DIS
LIN {X 144.015,Y -21.431,Z -159.525,A -90.000,B 90.000,C 0.000} C_DIS
LIN {X 111.857,Y -21.431,Z -159.525,A -90.000,B 90.000,C 0.000} C_DIS
LIN {X 111.545,Y -21.431,Z -163.301,A -90.000,B 90.000,C 0.000} C_DIS
LIN {X 111.195,Y -21.431,Z -167.073,A -90.000,B 90.000,C 0.000} C_DIS
LIN {X 144.015,Y -21.431,Z -167.073,A -90.000,B 90.000,C 0.000} C_DIS
LIN {X 144.015,Y -21.431,Z -174.622,A -90.000,B 90.000,C 0.000} C_DIS
LIN {X 110.376,Y -21.431,Z -174.622,A -90.000,B 90.000,C 0.000} C_DIS
LIN {X 109.907,Y -21.431,Z -178.399,A -90.000,B 90.000,C 0.000} C_DIS
LIN {X 109.399,Y -21.431,Z -182.171,A -90.000,B 90.000,C 0.000} C_DIS
LIN {X 144.015,Y -21.431,Z -182.171,A -90.000,B 90.000,C 0.000} C_DIS
LIN {X 144.015,Y -21.431,Z -189.720,A -90.000,B 90.000,C 0.000} C_DIS
LIN {X 108.264,Y -21.431,Z -189.720,A -90.000,B 90.000,C 0.000} C_DIS
LIN {X 107.636,Y -21.431,Z -193.498,A -90.000,B 90.000,C 0.000} C_DIS
LIN {X 106.969,Y -21.431,Z -197.269,A -90.000,B 90.000,C 0.000} C_DIS
LIN {X 144.015,Y -21.431,Z -197.269,A -90.000,B 90.000,C 0.000} C_DIS
LIN {X 144.015,Y -21.431,Z -204.817,A -90.000,B 90.000,C 0.000} C_DIS
LIN {X 105.512,Y -21.431,Z -204.817,A -90.000,B 90.000,C 0.000} C_DIS
LIN {X 104.721,Y -21.431,Z -208.596,A -90.000,B 90.000,C 0.000} C_DIS
LIN {X 103.892,Y -21.431,Z -212.366,A -90.000,B 90.000,C 0.000} C_DIS
LIN {X 144.015,Y -21.431,Z -212.366,A -90.000,B 90.000,C 0.000} C_DIS
LIN {X 144.015,Y -21.431,Z -219.915,A -90.000,B 90.000,C 0.000} C_DIS
LIN {X 102.122,Y -21.431,Z -219.915,A -90.000,B 90.000,C 0.000} C_DIS
LIN {X 101.534,Y -21.431,Z -222.438,A -90.000,B 90.000,C 0.000} C_DIS
LIN {X 100.918,Y -21.431,Z -224.954,A -90.000,B 90.000,C 0.000} C_DIS
LIN {X 100.275,Y -21.431,Z -227.464,A -90.000,B 90.000,C 0.000} C_DIS
LIN {X 144.015,Y -21.431,Z -227.464,A -90.000,B 90.000,C 0.000} C_DIS
LIN {X 144.015,Y -21.431,Z -235.012,A -90.000,B 90.000,C 0.000} C_DIS
LIN {X 98.161,Y -21.431,Z -235.012,A -90.000,B 90.000,C 0.000} C_DIS
LIN {X 97.393,Y -21.431,Z -237.537,A -90.000,B 90.000,C 0.000} C_DIS
LIN {X 96.597,Y -21.431,Z -240.054,A -90.000,B 90.000,C 0.000} C_DIS
LIN {X 95.773,Y -21.431,Z -242.561,A -90.000,B 90.000,C 0.000} C_DIS
LIN {X 144.015,Y -21.431,Z -242.561,A -90.000,B 90.000,C 0.000} C_DIS
LIN {X 145.015,Y -21.431,Z -243.561,A -90.000,B 90.000,C 0.000} C_DIS
LIN {X 145.015,Y -21.431,Z 0.000,A -90.000,B 90.000,C 0.000} C_DIS
LIN {X -145.015,Y -21.431,Z 0.000,A -90.000,B 90.000,C 0.000} C_DIS
LIN {X -145.015,Y -21.431,Z -243.561,A -90.000,B 90.000,C 0.000} C_DIS
LIN {X -123.357,Y -21.431,Z -243.561,A -90.000,B 90.000,C 0.000} C_DIS
LIN {X -120.017,Y -21.431,Z -241.310,A -90.000,B 90.000,C 0.000} C_DIS
LIN {X -116.697,Y -21.431,Z -239.030,A -90.000,B 90.000,C 0.000} C_DIS
